// TIA Portal V18 program export: 1 tag tables, 7 data types, 4 data blocks, 9 code blocks (in call order from the OBs), 2 instance data blocks

VAR_GLOBAL   // PLC tag table "Default tag table"
   D_INPUT AT %I0.0 : "DI";
   A_IN AT %I100.0 : "AI";
   RTD_IN AT %I108.0 : "RTD";
   D_OUTPUT AT %Q0.0 : "DO";
   A_OUT AT %Q100.0 : "AO";
   System_Byte AT %MB1 : Byte;
   FirstScan AT %M1.0 : Bool;
   DiagStatusUpdate AT %M1.1 : Bool;
   AlwaysTRUE AT %M1.2 : Bool;
   AlwaysFALSE AT %M1.3 : Bool;
   Clock_Byte AT %MB0 : Byte;
   Clock_10Hz AT %M0.0 : Bool;
   Clock_5Hz AT %M0.1 : Bool;
   "Clock_2.5Hz" AT %M0.2 : Bool;
   Clock_2Hz AT %M0.3 : Bool;
   "Clock_1.25Hz" AT %M0.4 : Bool;
   Clock_1Hz AT %M0.5 : Bool;
   "Clock_0.625Hz" AT %M0.6 : Bool;
   "Clock_0.5Hz" AT %M0.7 : Bool;
   Tag_1 AT %M5.0 : Bool;
   Tag_2 AT %M55.0 : Bool;
   Tag_3 AT %M75.0 : Bool;
END_VAR
VAR_GLOBAL CONSTANT   // user constants
   "None(2)" : Pip := 65535;
   "Automatic update(2)" : Pip := 0;
   "PIP 1(2)" : Pip := 1;
   "PIP 2(2)" : Pip := 2;
   "PIP 3(2)" : Pip := 3;
   "PIP 4(2)" : Pip := 4;
   "PIP 5" : Pip := 5;
   "PIP 6" : Pip := 6;
   "PIP 7" : Pip := 7;
   "PIP 8" : Pip := 8;
   "PIP 9" : Pip := 9;
   "PIP 10" : Pip := 10;
   "PIP 11" : Pip := 11;
   "PIP 12" : Pip := 12;
   "PIP 13" : Pip := 13;
   "PIP 14" : Pip := 14;
   "PIP 15" : Pip := 15;
   "PIP 16" : Pip := 16;
   "PIP 17" : Pip := 17;
   "PIP 18" : Pip := 18;
   "PIP 19" : Pip := 19;
   "PIP 20" : Pip := 20;
   "PIP 21" : Pip := 21;
   "PIP 22" : Pip := 22;
   "PIP 23" : Pip := 23;
   "PIP 24" : Pip := 24;
   "PIP 25" : Pip := 25;
   "PIP 26" : Pip := 26;
   "PIP 27" : Pip := 27;
   "PIP 28" : Pip := 28;
   "PIP 29" : Pip := 29;
   "PIP 30" : Pip := 30;
   "PIP 31" : Pip := 31;
   "PIP OB Servo(2)" : Pip := 32768;
   "Local~MC(2)" : Hw_SubModule := 51;
   "Local~Common(2)" : Hw_SubModule := 50;
   "Local~Device(2)" : Hw_Device := 32;
   "Local~Configuration(2)" : Hw_SubModule := 33;
   "Local~Display" : Hw_SubModule := 54;
   "Local~Exec(2)" : Hw_SubModule := 52;
   "Local(2)" : Hw_SubModule := 49;
   "Local~PROFINET_interface_1(2)" : Hw_Interface := 64;
   "Local~PROFINET_interface_1~Port_1(2)" : Hw_Interface := 65;
   "Local~PROFINET_interface_1~Port_2" : Hw_Interface := 66;
   "Local~Virtual_communication_interface" : Hw_Interface := 135;
   "Local~License_Manager" : Hw_SubModule := 42;
   "OB_Main(2)" : OB_PCYCLE := 1;
END_VAR

TYPE "AI"
// stored: IsFailsafeCompliant false
   STRUCT
      "FLOW METER" : Int;
      "CONDUCTIVITY METER" : Int;
      "SPARE AI1" : Int;
      "SPARE AI2" : Int;
   END_STRUCT;
END_TYPE

TYPE "AM CTRL"
// stored: IsFailsafeCompliant false
   STRUCT
      "AUTO/MAN" : Bool := TRUE;
      "MAN START" : Bool;
      "MAN STOP" : Bool;
   END_STRUCT;
END_TYPE

TYPE "AO"
// stored: IsFailsafeCompliant false
   STRUCT
      VFD : Int;
      "SPARE AO" : Int;
   END_STRUCT;
END_TYPE

TYPE "DI"
// stored: IsFailsafeCompliant false
   STRUCT
      START : Bool;
      STOP : Bool;
      EMERGENCY : Bool;
      ACKNOWLEDGE : Bool;
      "AUTO/MANUAL" : Bool;
      "RECUPARATION TANK HL" : Bool;
      "RECUPARATION TANK LL" : Bool;
      "HOT WATER TANK HL" : Bool;
      "HOT WATER TANK LL" : Bool;
      "CAUSTIC TANK HL" : Bool;
      "CAUSTIC TANK LL" : Bool;
      "ACID TANK HL" : Bool;
      "ACID TANK LL" : Bool;
      "SUPPLY PUMP RUN (VFD)" : Bool;
      RESERVED : Bool;
      RESERVED_1 : Bool;
      "SUPPLY PUMP TRIP (VFD)" : Bool;
      "ACID DOSING PUMP RUN" : Bool;
      "ACID DOSING PUMP TRIP" : Bool;
      "CAUSTIC DOSING PUMP RUN" : Bool;
      "CAUSTIC DOSING PUMP TRIP" : Bool;
      "RETURN PUMP 1 RUN" : Bool;
      "RETURN PUMP 1 TRIP" : Bool;
      "RETURN PUMP 2 RUN" : Bool;
      "RETURN PUMP 2 TRIP" : Bool;
      "RETURN PUMP 3 RUN" : Bool;
      "RETURN PUMP 3 TRIP" : Bool;
      "FLOW SWITCH" : Bool;
      "PRESSURE SWITCH" : Bool;
      SPARE_1 : Bool;
      SPARE_2 : Bool;
      SPARE_3 : Bool;
   END_STRUCT;
END_TYPE

TYPE "DO"
// stored: IsFailsafeCompliant false
   STRUCT
      BUZZER : Bool;
      "BFV 1" : Bool;
      "BFV 2" : Bool;
      "BFV 3" : Bool;
      "BFV 4" : Bool;
      "BFV 5" : Bool;
      "BFV 6" : Bool;
      "BFV 7" : Bool;
      "BFV 8" : Bool;
      "BFV 9" : Bool;
      R1 : Bool;
      R2 : Bool;
      R3 : Bool;
      R4 : Bool;
      R5 : Bool;
      R6 : Bool;
      "BFV 10" : Bool;
      "BFV 11" : Bool;
      "BFV 12" : Bool;
      "BFV 13" : Bool;
      "BFV 14" : Bool;
      "BFV 15" : Bool;
      "BFV 16" : Bool;
      "BFV 17" : Bool;
      "BFV 18" : Bool;
      "BFV 19" : Bool;
      "CIP SUPPLY PUMP START (VFD)" : Bool;
      "ACID DOSING PUMP" : Bool;
      "CAUSTIC DOSING PUMP" : Bool;
      "RETURN PUMP 1" : Bool;
      "RETURN PUMP 2" : Bool;
      "RETUEN PUMP 3" : Bool;
   END_STRUCT;
END_TYPE

TYPE "RTD"
// stored: IsFailsafeCompliant false
   STRUCT
      "RECUPERATION TANK" : Int;
      "HOT WATER TANK" : Int;
      "CAUSTIC TANK" : Int;
      "ACID TANK" : Int;
      "FWD LINE" : Int;
      "RETURN LINE" : Int;
      "SPARE RTD" : Int;
      "SPARE RTD 1" : Int;
   END_STRUCT;
END_TYPE

TYPE "TANK DATA"
// stored: IsFailsafeCompliant false
   STRUCT
      "TANK TEMP SP" : Real;
      "LINE TEMP SP" : Real;
      "RETURN SP" : Real;
      "COND SP" : Real;
      "HYSTERIRIS TEMP" : Real;
      "HYSTERISIS COND" : Real;
      "CYCLE TIME MIN" : Int;
      "CYCLE TIME SEC" : Int;
      "ELAPSED MIN" : Int;
      "ELAPSED SEC" : Int;
   END_STRUCT;
END_TYPE

DATA_BLOCK "HMI ALARM DB"   // DB5
{ S7_Optimized_Access := 'FALSE' }
VERSION : 0.1
// stored: AutoNumber true, DBAccessibleFromOPCUA true, IsOnlyStoredInLoadMemory false, IsWriteProtectedInAS false
   VAR
      "FEED PUMP" : Byte;   // XO- INTERLOCK
      "ACID DOSING" : Byte;   // X1 - TRIP
      "CAUSTIC DOSING" : Byte;   // X2 - RUN FB ERROR
      "RP 1" : Byte;
      "RP 2" : Byte;
      "RP 3" : Byte;
      "RETURN NOT SELECTED" : Bool;
      "CYCLE NOT SELECTED" : Bool;
      "WATER FLUSH TIME NOT SET" : Bool;
      "HOT WATER TIME NOT SET" : Bool;
      "RECUP TIME NOT SET" : Bool;
      "ACIDIC TIME NOT SET" : Bool;
      "CAUSTIC TIMENOT SET" : Bool;
   END_VAR
BEGIN
END_DATA_BLOCK

DATA_BLOCK "HMI DB"   // DB2
{ S7_Optimized_Access := 'FALSE' }
VERSION : 0.1
// stored: AutoNumber true, DBAccessibleFromOPCUA true, IsOnlyStoredInLoadMemory false, IsWriteProtectedInAS false
   VAR RETAIN
      "START PREP" : Bool := FALSE;
      "START CIP" : Bool := FALSE;
      "CIP 3 STEP" : Bool := FALSE;
      "CIP 5 STEP" : Bool := FALSE;
      "CIP 7 STEP" : Bool := FALSE;
      RP1 : Bool;
      RP2 : Bool;
      RP3 : Bool;
      "RESUME CIP" : Bool;
      "RP1 SELECTED" : Bool;
      "RP2 SELECTED" : Bool;
      "RP3 SELECTED" : Bool;
      "3 STEP STATUS" : Word;
      "5 STEP STATUS" : Word;
      "9 STEP STATUS" : Word;
      RESERVE : Array[0..28] of Word;
      "BFV1 AM" { S7_SetPoint := 'True'} : "AM CTRL";
      "BFV2 AM" { S7_SetPoint := 'True'} : "AM CTRL";
      "BFV3 AM" { S7_SetPoint := 'True'} : "AM CTRL";
      "BFV4 AM" { S7_SetPoint := 'True'} : "AM CTRL";
      "BFV5 AM" { S7_SetPoint := 'True'} : "AM CTRL";
      "BFV6 AM" { S7_SetPoint := 'True'} : "AM CTRL";
      "BFV7 AM" { S7_SetPoint := 'True'} : "AM CTRL";
      "BFV8 AM" { S7_SetPoint := 'True'} : "AM CTRL";
      "BFV9 AM" { S7_SetPoint := 'True'} : "AM CTRL";
      "BFV10 AM" { S7_SetPoint := 'True'} : "AM CTRL";
      "BFV11 AM" { S7_SetPoint := 'True'} : "AM CTRL";
      "BFV12 AM" { S7_SetPoint := 'True'} : "AM CTRL";
      "BFV13 AM" { S7_SetPoint := 'True'} : "AM CTRL";
      "BFV14 AM" { S7_SetPoint := 'True'} : "AM CTRL";
      "BFV15 AM" { S7_SetPoint := 'True'} : "AM CTRL";
      "BFV16 AM" { S7_SetPoint := 'True'} : "AM CTRL";
      "BFV17 AM" { S7_SetPoint := 'True'} : "AM CTRL";
      "BFV18 AM" { S7_SetPoint := 'True'} : "AM CTRL";
      "BFV19 AM" { S7_SetPoint := 'True'} : "AM CTRL";
      "VFD AM" { S7_SetPoint := 'True'} : "AM CTRL";
      "RETURN PUMP 1 AM" { S7_SetPoint := 'True'} : "AM CTRL";
      "RETURN PUMP 2 AM" { S7_SetPoint := 'True'} : "AM CTRL";
      "RETURN PUMP 3 AM" { S7_SetPoint := 'True'} : "AM CTRL";
      "CAUSTIC AM" { S7_SetPoint := 'True'} : "AM CTRL";
      "ACIDIC AM" { S7_SetPoint := 'True'} : "AM CTRL";
      "PUMP SLOW SP" : Int := 0;
      RECUP : "TANK DATA";
      "HOT WATER" : "TANK DATA";
      CAUSTIC : "TANK DATA";
      ACIDIC : "TANK DATA";
      "ANALOG VALUES" : Struct
         FLOW : Real := 0.0;
         CONDCTIVITY : Real := 0.0;
         "RECUP TEMP" : Real := 0.0;
         "HOT WTR TEMP" : Real := 0.0;
         "CAUSTIC TEMP" : Real := 0.0;
         "ACID TEMP" : Real := 0.0;
         "RETURN LINE TEMP" : Real := 0.0;
      END_STRUCT;
      "START DELAYS" : Struct
         "RP1 MIN" : Int;
         "RP1 SEC" : Int;
         "RP2 MIN" : Int;
         "RP2 SEC" : Int;
         "RP3 MIN" : Int;
         "RP3 SEC" : Int;
      END_STRUCT;
      "COMMON SETPOINTS" : Struct   // 286
         "COND MIN FOR RECUP" : Real;
         "TMP MIN FOR RECUP" : Real;
         "WATER FLUSH MIN" : Int;
         "WATER FLUSH SEC" : Int;
         "WATER FLUSH REM MIN" : Int;
         "WATER FLUSH REM SEC" : Int;
      END_STRUCT;
      "Fwd line temp" : Real;
   END_VAR
BEGIN
   "BFV1 AM"."AUTO/MAN" := TRUE;
   "BFV1 AM"."MAN START" := FALSE;
   "BFV1 AM"."MAN STOP" := FALSE;
   "BFV2 AM"."AUTO/MAN" := TRUE;
   "BFV2 AM"."MAN START" := FALSE;
   "BFV2 AM"."MAN STOP" := FALSE;
   "BFV3 AM"."AUTO/MAN" := TRUE;
   "BFV3 AM"."MAN START" := FALSE;
   "BFV3 AM"."MAN STOP" := FALSE;
   "BFV4 AM"."AUTO/MAN" := TRUE;
   "BFV4 AM"."MAN START" := FALSE;
   "BFV4 AM"."MAN STOP" := FALSE;
   "BFV5 AM"."AUTO/MAN" := TRUE;
   "BFV5 AM"."MAN START" := FALSE;
   "BFV5 AM"."MAN STOP" := FALSE;
   "BFV6 AM"."AUTO/MAN" := TRUE;
   "BFV6 AM"."MAN START" := FALSE;
   "BFV6 AM"."MAN STOP" := FALSE;
   "BFV7 AM"."AUTO/MAN" := TRUE;
   "BFV7 AM"."MAN START" := FALSE;
   "BFV7 AM"."MAN STOP" := FALSE;
   "BFV8 AM"."AUTO/MAN" := TRUE;
   "BFV8 AM"."MAN START" := FALSE;
   "BFV8 AM"."MAN STOP" := FALSE;
   "BFV9 AM"."AUTO/MAN" := TRUE;
   "BFV9 AM"."MAN START" := FALSE;
   "BFV9 AM"."MAN STOP" := FALSE;
   "BFV10 AM"."AUTO/MAN" := TRUE;
   "BFV10 AM"."MAN START" := FALSE;
   "BFV10 AM"."MAN STOP" := FALSE;
   "BFV11 AM"."AUTO/MAN" := TRUE;
   "BFV11 AM"."MAN START" := FALSE;
   "BFV11 AM"."MAN STOP" := FALSE;
   "BFV12 AM"."AUTO/MAN" := TRUE;
   "BFV12 AM"."MAN START" := FALSE;
   "BFV12 AM"."MAN STOP" := FALSE;
   "BFV13 AM"."AUTO/MAN" := TRUE;
   "BFV13 AM"."MAN START" := FALSE;
   "BFV13 AM"."MAN STOP" := FALSE;
   "BFV14 AM"."AUTO/MAN" := TRUE;
   "BFV14 AM"."MAN START" := FALSE;
   "BFV14 AM"."MAN STOP" := FALSE;
   "BFV15 AM"."AUTO/MAN" := TRUE;
   "BFV15 AM"."MAN START" := FALSE;
   "BFV15 AM"."MAN STOP" := FALSE;
   "BFV16 AM"."AUTO/MAN" := TRUE;
   "BFV16 AM"."MAN START" := FALSE;
   "BFV16 AM"."MAN STOP" := FALSE;
   "BFV17 AM"."AUTO/MAN" := TRUE;
   "BFV17 AM"."MAN START" := FALSE;
   "BFV17 AM"."MAN STOP" := FALSE;
   "BFV18 AM"."AUTO/MAN" := TRUE;
   "BFV18 AM"."MAN START" := FALSE;
   "BFV18 AM"."MAN STOP" := FALSE;
   "BFV19 AM"."AUTO/MAN" := TRUE;
   "BFV19 AM"."MAN START" := FALSE;
   "BFV19 AM"."MAN STOP" := FALSE;
   "VFD AM"."AUTO/MAN" := TRUE;
   "VFD AM"."MAN START" := FALSE;
   "VFD AM"."MAN STOP" := FALSE;
   "RETURN PUMP 1 AM"."AUTO/MAN" := TRUE;
   "RETURN PUMP 1 AM"."MAN START" := FALSE;
   "RETURN PUMP 1 AM"."MAN STOP" := FALSE;
   "RETURN PUMP 2 AM"."AUTO/MAN" := TRUE;
   "RETURN PUMP 2 AM"."MAN START" := FALSE;
   "RETURN PUMP 2 AM"."MAN STOP" := FALSE;
   "RETURN PUMP 3 AM"."AUTO/MAN" := TRUE;
   "RETURN PUMP 3 AM"."MAN START" := FALSE;
   "RETURN PUMP 3 AM"."MAN STOP" := FALSE;
   "CAUSTIC AM"."AUTO/MAN" := TRUE;
   "CAUSTIC AM"."MAN START" := FALSE;
   "CAUSTIC AM"."MAN STOP" := FALSE;
   "ACIDIC AM"."AUTO/MAN" := TRUE;
   "ACIDIC AM"."MAN START" := FALSE;
   "ACIDIC AM"."MAN STOP" := FALSE;
   RECUP."COND SP" := 0.0;
   RECUP."HYSTERIRIS TEMP" := 0.0;
   RECUP."HYSTERISIS COND" := 0.0;
   RECUP."CYCLE TIME SEC" := 0;
   RECUP."ELAPSED MIN" := 0;
   RECUP."ELAPSED SEC" := 0;
   "HOT WATER"."COND SP" := 0.0;
   "HOT WATER"."HYSTERIRIS TEMP" := 0.0;
   "HOT WATER"."HYSTERISIS COND" := 0.0;
   "HOT WATER"."CYCLE TIME MIN" := 0;
   "HOT WATER"."CYCLE TIME SEC" := 0;
   "HOT WATER"."ELAPSED MIN" := 0;
   "HOT WATER"."ELAPSED SEC" := 0;
   CAUSTIC."COND SP" := 0.0;
   CAUSTIC."HYSTERIRIS TEMP" := 0.0;
   CAUSTIC."HYSTERISIS COND" := 0.0;
   CAUSTIC."CYCLE TIME MIN" := 0;
   CAUSTIC."CYCLE TIME SEC" := 0;
   CAUSTIC."ELAPSED MIN" := 0;
   CAUSTIC."ELAPSED SEC" := 0;
   ACIDIC."COND SP" := 0.0;
   ACIDIC."HYSTERIRIS TEMP" := 0.0;
   ACIDIC."HYSTERISIS COND" := 0.0;
   ACIDIC."CYCLE TIME MIN" := 0;
   ACIDIC."CYCLE TIME SEC" := 0;
   ACIDIC."ELAPSED MIN" := 0;
   ACIDIC."ELAPSED SEC" := 0;
END_DATA_BLOCK

DATA_BLOCK "IO_MAP"   // DB1
{ S7_Optimized_Access := 'FALSE' }
VERSION : 0.1
// stored: AutoNumber true, DBAccessibleFromOPCUA true, IsOnlyStoredInLoadMemory false, IsWriteProtectedInAS false
   VAR
      D_IN { S7_SetPoint := 'True'} : "DI";
      D_OUT { S7_SetPoint := 'True'} : "DO";
      A_OUT { S7_SetPoint := 'True'} : "AO";
      A_IN { S7_SetPoint := 'True'} : "AI";
      RTD { S7_SetPoint := 'True'} : "RTD";
   END_VAR
BEGIN
END_DATA_BLOCK

DATA_BLOCK "OPERATIONS DB"   // DB3
{ S7_Optimized_Access := 'TRUE' }
VERSION : 0.1
// stored: AutoNumber true, DBAccessibleFromOPCUA true, IsOnlyStoredInLoadMemory false, IsRetainMemResEnabled false, IsWriteProtectedInAS false, MemoryReserve 100
   VAR
      "SYSTEM STARTED" : Bool;
   END_VAR
BEGIN
END_DATA_BLOCK

ORGANIZATION_BLOCK "Main"   // OB1, LAD, ProgramCycle
TITLE = "Main Program Sweep (Cycle)"
{ S7_Optimized_Access := 'TRUE' }
VERSION : 0.1
// stored: AutoNumber true, IsIECCheckEnabled false, SetENOAutomatically false
   VAR_INPUT
      Initial_Call : Bool;   // Initial call of this OB
      Remanence : Bool;   // =True, if remanent data are available
   END_VAR
   VAR_TEMP   // added for the SCL form of the ladder/FBD networks
      _w1 : Bool;
   END_VAR
BEGIN

REGION Network 1
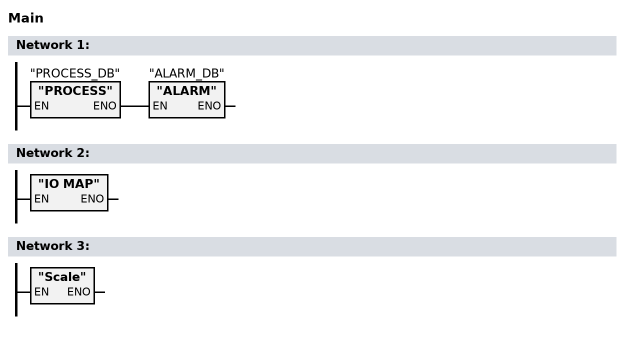
   RUNG wire#powerrail
      "PROCESS_DB"()
      "ALARM_DB"()
   END_RUNG
   // the same network as SCL:
   "PROCESS_DB"(ENO => #_w1);   // "PROCESS"
   IF #_w1 THEN
       "ALARM_DB"();   // "ALARM"
   END_IF;
END_REGION

REGION Network 2
   RUNG wire#powerrail
      "IO MAP"()
   END_RUNG
   // the same network as SCL:
   "IO MAP"();
END_REGION

REGION Network 3
   RUNG wire#powerrail
      "Scale"()
   END_RUNG
   // the same network as SCL:
   "Scale"();
END_REGION
END_ORGANIZATION_BLOCK

FUNCTION_BLOCK "PROCESS"   // FB3, LAD
{ S7_Optimized_Access := 'TRUE' }
VERSION : 0.1
// stored: AutoNumber true, IsIECCheckEnabled false, IsRetainMemResEnabled false, MemoryReserve 100, SetENOAutomatically false, UDAEnableTagReadback false
   VAR
      "RECUP TANK" { S7_SetPoint := 'True'} : "TANK";
      "HOT WATER TANK" { S7_SetPoint := 'True'} : "TANK";
      "CAUSTIC TANK" { S7_SetPoint := 'True'} : "TANK";
      "ACID TANK" { S7_SetPoint := 'True'} : "TANK";
      "RECUP PREP DONE" { S7_SetPoint := 'True'} : Bool;
      "HOT WTR PREP DONE" : Bool;
      "CAUSTIC PREP DONE" : Bool;
      "ACID PREP DONE" : Bool;
      "PREP FINISHED PULSE" : Bool;
      P1 : Bool;
      P2 : Bool;
      P3 : Bool;
      P4 : Bool;
      P5 : Bool;
      P6 : Bool;
      P7 : Bool;
      P8 : Bool;
      P9 : Bool;
      P10 : Bool;
      CIP_STARTED : Bool;
      "3 CIP FINISH PULSE" : Bool;
      "5 CIP FINISH PULSE" : Bool;
      "7 CIP FINISH PULSE" : Bool;
      "PUMP OK" : Bool;
   END_VAR
   VAR RETAIN
      "RECUP CIP DONE" : Array[0..4] of Bool;
      "HOT WTR CIP DONE" : Array[0..4] of Bool;
      "CAUSTIC CIP DONE" : Array[0..4] of Bool;
      "ACID CIP DONE" : Array[0..4] of Bool;
      "WATER FLUSH CIP DONE" : Array[0..4] of Bool;
      "CIP_STEP SELECTED" : Int;
   END_VAR
   VAR
      "CURCULATION PUMP" { S7_SetPoint := 'True'} : "PUMP";
      "BFV1 CTRL" { S7_SetPoint := 'True'} : "VALVE CTRL";
      "BFV2 CTRL" { S7_SetPoint := 'True'} : "VALVE CTRL";
      "BFV3 CTRL" { S7_SetPoint := 'True'} : "VALVE CTRL";
      "BFV4 CTRL" { S7_SetPoint := 'True'} : "VALVE CTRL";
      "BFV5 CTRL" { S7_SetPoint := 'True'} : "VALVE CTRL";
      "BFV6 CTRL" { S7_SetPoint := 'True'} : "VALVE CTRL";
      "BFV7 CTRL" { S7_SetPoint := 'True'} : "VALVE CTRL";
      "BFV8 CTRL" { S7_SetPoint := 'True'} : "VALVE CTRL";
      "BFV9 CTRL" { S7_SetPoint := 'True'} : "VALVE CTRL";
      "BFV10 CTRL" { S7_SetPoint := 'True'} : "VALVE CTRL";
      "BFV11 CTRL" { S7_SetPoint := 'True'} : "VALVE CTRL";
      "BFV12 CTRL" { S7_SetPoint := 'True'} : "VALVE CTRL";
      "BFV13 CTRL" { S7_SetPoint := 'True'} : "VALVE CTRL";
      "BFV14 CTRL" { S7_SetPoint := 'True'} : "VALVE CTRL";
      "BFV15 CTRL" { S7_SetPoint := 'True'} : "VALVE CTRL";
      "BFV16 CTRL" { S7_SetPoint := 'True'} : "VALVE CTRL";
      "BFV17 CTRL" { S7_SetPoint := 'True'} : "VALVE CTRL";
      "BFV18 CTRL" { S7_SetPoint := 'True'} : "VALVE CTRL";
      "BFV19 CTRL" { S7_SetPoint := 'True'} : "VALVE CTRL";
      "BFV20 CTRL" { S7_SetPoint := 'True'} : "VALVE CTRL";
      "CAUSTIC DOSING" { S7_SetPoint := 'True'} : "PUMP";
      "ACID DOSING" { S7_SetPoint := 'True'} : "PUMP";
      "RETURN PUMP 1" { S7_SetPoint := 'True'} : "PUMP";
      "RETURN PUMP 2" { S7_SetPoint := 'True'} : "PUMP";
      "RETURN PUMP 3" { S7_SetPoint := 'True'} : "PUMP";
      "WATER FLUSH" { S7_SetPoint := 'True'} : TON_TIME;
   END_VAR
   VAR_TEMP
      "RECUP PREP START" : Bool;
      "RECUP CIP START" : Bool;
      "HOT WTR PREP START" : Bool;
      "HOT WTR CIP START" : Bool;
      "CAUSTIC PREP START" : Bool;
      "CAUSTIC CIP START" : Bool;
      "ACID PREP START" : Bool;
      "ACID CIP START" : Bool;
      "WATER FLUSH CIP START" : Bool;
      "RP1 START" : Bool;
      "RP2 START" : Bool;
      "RP3 START" : Bool;
      CIRCULATION : Bool;
      "WF PT" : Time;
      "WF ET" : Time;
      RECUP : Struct
         "INLET 1 OPEN" : Bool;
         "INLET 2 OPEN" : Bool;
         "OUTLE OPEN" : Bool;
         "START DOZING" : Bool;
         FLUSH : Bool;
         HEATING : Bool;
         "PREP DONE" : Bool;
      END_STRUCT;
      HTWTR : Struct
         "INLET 1 OPEN" : Bool;
         "INLET 2 OPEN" : Bool;
         "OUTLE OPEN" : Bool;
         "START DOZING" : Bool;
         FLUSH : Bool;
         HEATING : Bool;
         "PREP DONE" : Bool;
      END_STRUCT;
      CAUSTIC : Struct
         "INLET 1 OPEN" : Bool;
         "INLET 2 OPEN" : Bool;
         "OUTLE OPEN" : Bool;
         "START DOZING" : Bool;
         FLUSH : Bool;
         HEATING : Bool;
         "PREP DONE" : Bool;
      END_STRUCT;
      ACIDIC : Struct
         "INLET 1 OPEN" : Bool;
         "INLET 2 OPEN" : Bool;
         "OUTLE OPEN" : Bool;
         "START DOZING" : Bool;
         FLUSH : Bool;
         HEATING : Bool;
         "PREP DONE" : Bool;
      END_STRUCT;
      "TEMP ARRAY" : Array[0..4] of Bool;
      "CYCLE SELECTED" : Bool;
      "RETURN SELECTED" : Bool;
      "settings OK" : Bool;
      "WATER TIME OK" : Bool;
      "CAUSTIC TIME OK" : Bool;
      "HOTWATER TIME OK" : Bool;
      "REUP TIME OK" : Bool;
      "ACID TIME OK" : Bool;
   END_VAR
   VAR_TEMP   // added for the SCL form of the ladder/FBD networks
      _w1 : Bool;
      _w2 : Bool;
      _w3 : Bool;
      _w4 : Bool;
      _w5 : Bool;
      _w6 : Bool;
      _w7 : Bool;
      _w8 : Bool;
      _w9 : Bool;
      _w10 : Bool;
   END_VAR
BEGIN

REGION Network 1: START PREP
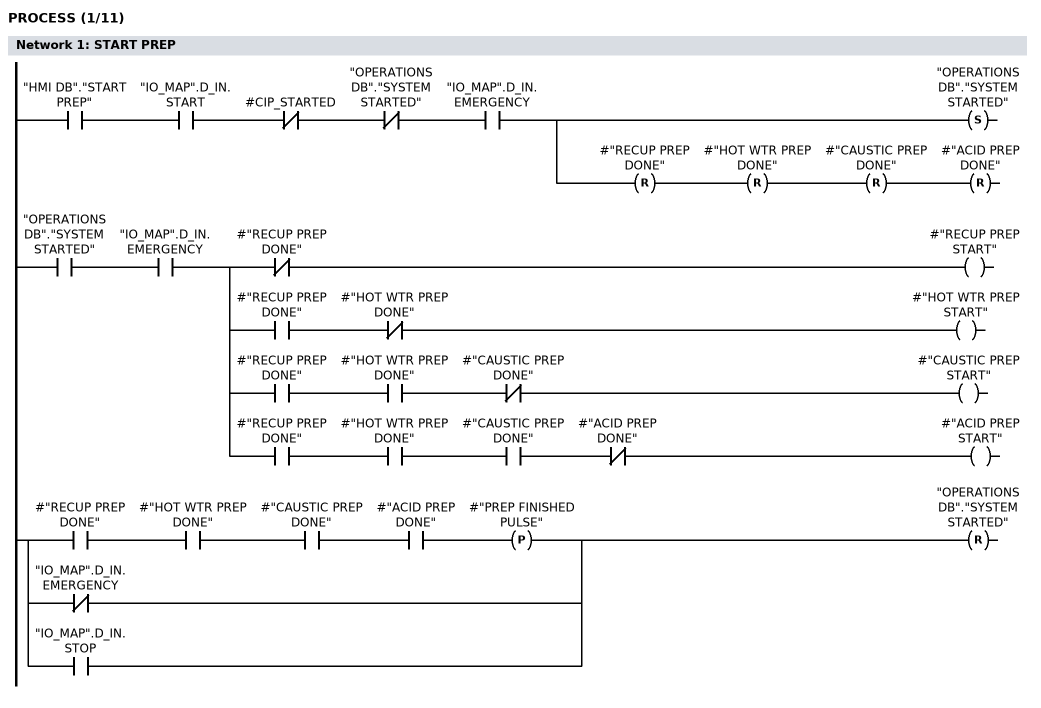
   RUNG wire#powerrail
      Contact( "HMI DB"."START PREP" )
      Contact( "IO_MAP".D_IN.START )
      I_Contact( #CIP_STARTED )
      I_Contact( "OPERATIONS DB"."SYSTEM STARTED" )
      Contact( "IO_MAP".D_IN.EMERGENCY )
      wire#w1
      S_Coil( "OPERATIONS DB"."SYSTEM STARTED" )
   END_RUNG
   RUNG wire#w1
      R_Coil( #"RECUP PREP DONE" )
      R_Coil( #"HOT WTR PREP DONE" )
      R_Coil( #"CAUSTIC PREP DONE" )
      R_Coil( #"ACID PREP DONE" )
   END_RUNG
   RUNG wire#powerrail
      Contact( "OPERATIONS DB"."SYSTEM STARTED" )
      Contact( "IO_MAP".D_IN.EMERGENCY )
      wire#w2
      I_Contact( #"RECUP PREP DONE" )
      Coil( #"RECUP PREP START" )
   END_RUNG
   RUNG wire#w2
      Contact( #"RECUP PREP DONE" )
      I_Contact( #"HOT WTR PREP DONE" )
      Coil( #"HOT WTR PREP START" )
   END_RUNG
   RUNG wire#w2
      Contact( #"RECUP PREP DONE" )
      Contact( #"HOT WTR PREP DONE" )
      I_Contact( #"CAUSTIC PREP DONE" )
      Coil( #"CAUSTIC PREP START" )
   END_RUNG
   RUNG wire#w2
      Contact( #"RECUP PREP DONE" )
      Contact( #"HOT WTR PREP DONE" )
      Contact( #"CAUSTIC PREP DONE" )
      I_Contact( #"ACID PREP DONE" )
      Coil( #"ACID PREP START" )
   END_RUNG
   RUNG wire#powerrail
      Contact( #"RECUP PREP DONE" )
      Contact( #"HOT WTR PREP DONE" )
      Contact( #"CAUSTIC PREP DONE" )
      Contact( #"ACID PREP DONE" )
      P_Trig( #"PREP FINISHED PULSE" )
      wire#w3
      R_Coil( "OPERATIONS DB"."SYSTEM STARTED" )
   END_RUNG
   RUNG wire#powerrail
      I_Contact( "IO_MAP".D_IN.EMERGENCY )
   END_RUNG wire#w3
   RUNG wire#powerrail
      Contact( "IO_MAP".D_IN.STOP )
   END_RUNG wire#w3
   // the same network as SCL:
   #_w1 := "HMI DB"."START PREP" AND "IO_MAP".D_IN.START AND NOT #CIP_STARTED AND NOT "OPERATIONS DB"."SYSTEM STARTED" AND "IO_MAP".D_IN.EMERGENCY;
   IF #_w1 THEN
       "OPERATIONS DB"."SYSTEM STARTED" := TRUE;
       #"RECUP PREP DONE" := FALSE;
       #"HOT WTR PREP DONE" := FALSE;
       #"CAUSTIC PREP DONE" := FALSE;
       #"ACID PREP DONE" := FALSE;
   END_IF;
   #_w2 := "OPERATIONS DB"."SYSTEM STARTED" AND "IO_MAP".D_IN.EMERGENCY;
   #"RECUP PREP START" := #_w2 AND NOT #"RECUP PREP DONE";
   #"HOT WTR PREP START" := #_w2 AND #"RECUP PREP DONE" AND NOT #"HOT WTR PREP DONE";
   #"CAUSTIC PREP START" := #_w2 AND #"RECUP PREP DONE" AND #"HOT WTR PREP DONE" AND NOT #"CAUSTIC PREP DONE";
   #"ACID PREP START" := #_w2 AND #"RECUP PREP DONE" AND #"HOT WTR PREP DONE" AND #"CAUSTIC PREP DONE" AND NOT #"ACID PREP DONE";
   #_w3 := #"RECUP PREP DONE" AND #"HOT WTR PREP DONE" AND #"CAUSTIC PREP DONE" AND #"ACID PREP DONE";
   #_w4 := #_w3 AND NOT #"PREP FINISHED PULSE";   // rising edge
   #"PREP FINISHED PULSE" := #_w3;
   IF #_w4 OR NOT "IO_MAP".D_IN.EMERGENCY OR "IO_MAP".D_IN.STOP THEN
       "OPERATIONS DB"."SYSTEM STARTED" := FALSE;
   END_IF;
END_REGION

REGION Network 2 (SCL): START CIP
   //check for settings if it is ok to procced with CIP steps
   #"CYCLE SELECTED" := "HMI DB"."CIP 3 STEP" OR "HMI DB"."CIP 5 STEP" OR "HMI DB"."CIP 7 STEP";
   #"RETURN SELECTED" := "HMI DB"."RP1 SELECTED" OR "HMI DB"."RP2 SELECTED" OR "HMI DB"."RP3 SELECTED";
   #"WATER TIME OK" := ("HMI DB"."COMMON SETPOINTS"."WATER FLUSH MIN" > 0 OR "HMI DB"."COMMON SETPOINTS"."WATER FLUSH SEC" > 0);
   #"REUP TIME OK" := ("HMI DB".RECUP."CYCLE TIME MIN" > 0 OR "HMI DB".RECUP."CYCLE TIME SEC" > 0);
   #"HOTWATER TIME OK" := ("HMI DB"."HOT WATER"."CYCLE TIME MIN" > 0 OR "HMI DB"."HOT WATER"."CYCLE TIME SEC" > 0);
   #"CAUSTIC TIME OK" := ("HMI DB".CAUSTIC."CYCLE TIME MIN" > 0 OR "HMI DB".CAUSTIC."CYCLE TIME SEC" > 0) OR "HMI DB"."CIP 3 STEP";
   #"ACID TIME OK" := ("HMI DB".ACIDIC ."CYCLE TIME MIN" > 0 OR "HMI DB".ACIDIC."CYCLE TIME SEC" > 0) OR "HMI DB"."CIP 3 STEP" OR "HMI DB"."CIP 5 STEP" ;

   #"settings OK" := #"CYCLE SELECTED" AND #"RETURN SELECTED" AND #"WATER TIME OK" AND #"REUP TIME OK" AND #"HOTWATER TIME OK" AND #"CAUSTIC TIME OK" AND #"ACID TIME OK";
   //IF SETTINGS ARE OK STARTING CONDITIONS FOR CIP CYCLE
   IF ("HMI DB"."START CIP" OR "HMI DB"."RESUME CIP") AND"IO_MAP".D_IN.START AND"IO_MAP".D_IN.EMERGENCY AND NOT"OPERATIONS DB"."SYSTEM STARTED"AND NOT #CIP_STARTED AND NOT"IO_MAP".D_IN.STOP  AND #"settings OK" THEN
       #CIP_STARTED := TRUE;
       IF "HMI DB"."CIP 3 STEP" THEN
           #"CIP_STEP SELECTED" := 3;
       ELSIF "HMI DB"."CIP 5 STEP" THEN
           #"CIP_STEP SELECTED" := 5;
       ELSIF "HMI DB"."CIP 7 STEP" THEN
           #"CIP_STEP SELECTED" := 9;
       END_IF;
       IF "HMI DB"."START CIP" THEN
           #"RECUP CIP DONE" := #"TEMP ARRAY";
           #"HOT WTR CIP DONE" := #"TEMP ARRAY";
           #"CAUSTIC CIP DONE" := #"TEMP ARRAY";
           #"ACID CIP DONE" := #"TEMP ARRAY";
           #"WATER FLUSH CIP DONE" := #"TEMP ARRAY";
       END_IF;

       //STOP CONDITION IF EMERGENCY OR STOP IS PRESSED
   ELSIF NOT "IO_MAP".D_IN.EMERGENCY OR "IO_MAP".D_IN.STOP  THEN
       #CIP_STARTED := FALSE;
        #"CIP_STEP SELECTED" := 0;
   END_IF;
END_REGION

REGION Network 3 (SCL): CIP SEQUENCE
   IF #CIP_STARTED THEN
       CASE #"CIP_STEP SELECTED" OF
               //SEQUENCE FOR 3 STEP OPERATION
           3:
               #"RECUP CIP START" := NOT #"RECUP CIP DONE"[0];
               #"HOT WTR CIP START" := #"RECUP CIP DONE"[0] AND NOT #"HOT WTR CIP DONE"[0];
               #"WATER FLUSH CIP START" := #"RECUP CIP DONE"[0] AND #"HOT WTR CIP DONE"[0] AND NOT #"WATER FLUSH CIP DONE"[0];

               //3 STEP DONE CONDITION
               IF #"RECUP CIP DONE"[0] AND #"HOT WTR CIP DONE"[0] AND #"WATER FLUSH CIP DONE"[0] AND NOT #"3 CIP FINISH PULSE" THEN
                   #CIP_STARTED := FALSE;
                   #"3 CIP FINISH PULSE" := TRUE;
               ELSIF NOT (#"RECUP CIP DONE"[0] AND #"HOT WTR CIP DONE"[0] AND #"WATER FLUSH CIP DONE"[0]) THEN
                   #"3 CIP FINISH PULSE" := FALSE;
               END_IF;
           5:
               //SEQUENCE FOR 5 STEP OPERATION
               #"RECUP CIP START" := NOT #"RECUP CIP DONE"[0];
               #"CAUSTIC CIP START" := #"RECUP CIP DONE"[0] AND NOT #"CAUSTIC CIP DONE"[0];
               #"WATER FLUSH CIP START" := (#"RECUP CIP DONE"[0] AND #"CAUSTIC CIP DONE"[0] AND NOT #"WATER FLUSH CIP DONE"[0])
               OR (#"RECUP CIP DONE"[0] AND #"CAUSTIC CIP DONE"[0] AND #"WATER FLUSH CIP DONE"[0] AND #"HOT WTR CIP DONE"[0] AND NOT #"WATER FLUSH CIP DONE"[1]);
               #"HOT WTR CIP START" := #"RECUP CIP DONE"[0] AND #"CAUSTIC CIP DONE"[0] AND #"WATER FLUSH CIP DONE"[0] AND NOT #"HOT WTR CIP DONE"[0];

               // 5 STEP DONE CONDITION
               IF #"RECUP CIP DONE"[0] AND #"CAUSTIC CIP DONE"[0] AND #"WATER FLUSH CIP DONE"[0] AND #"HOT WTR CIP DONE"[0] AND #"WATER FLUSH CIP DONE"[1] AND NOT #"5 CIP FINISH PULSE" THEN
                   #CIP_STARTED := FALSE;
                   #"5 CIP FINISH PULSE" := TRUE;
               ELSIF NOT (#"RECUP CIP DONE"[0] AND #"CAUSTIC CIP DONE"[0] AND #"WATER FLUSH CIP DONE"[0] AND #"HOT WTR CIP DONE"[0] AND #"WATER FLUSH CIP DONE"[1]) THEN
                   #"5 CIP FINISH PULSE" := FALSE;
               END_IF;

           9:
               //SEQUENCE FOR 9 STEP OPERATION
               #"RECUP CIP START" := NOT #"RECUP CIP DONE"[0];

               #"CAUSTIC CIP START" := (#"RECUP CIP DONE"[0] AND NOT #"CAUSTIC CIP DONE"[0])
               OR #"RECUP CIP DONE"[0] AND #"CAUSTIC CIP DONE"[0] AND #"WATER FLUSH CIP DONE"[0] AND #"ACID CIP DONE"[0] AND #"WATER FLUSH CIP DONE"[1] AND NOT #"CAUSTIC CIP DONE"[1];

               #"WATER FLUSH CIP START" := (#"RECUP CIP DONE"[0] AND #"CAUSTIC CIP DONE"[0] AND NOT #"WATER FLUSH CIP DONE"[0])
               OR (#"RECUP CIP DONE"[0] AND #"CAUSTIC CIP DONE"[0] AND #"WATER FLUSH CIP DONE"[0] AND #"ACID CIP DONE"[0] AND NOT #"WATER FLUSH CIP DONE"[1])
               OR (#"RECUP CIP DONE"[0] AND #"CAUSTIC CIP DONE"[0] AND #"WATER FLUSH CIP DONE"[0] AND #"ACID CIP DONE"[0] AND #"WATER FLUSH CIP DONE"[1] AND #"CAUSTIC CIP DONE"[1] AND NOT #"WATER FLUSH CIP DONE"[2])
               OR (#"RECUP CIP DONE"[0] AND #"CAUSTIC CIP DONE"[0] AND #"WATER FLUSH CIP DONE"[0] AND #"ACID CIP DONE"[0] AND  #"WATER FLUSH CIP DONE"[1] AND #"CAUSTIC CIP DONE"[1] AND #"WATER FLUSH CIP DONE"[2] AND #"HOT WTR CIP DONE"[0] AND NOT #"WATER FLUSH CIP DONE"[3]);

               #"ACID CIP START" := #"RECUP CIP DONE"[0] AND #"CAUSTIC CIP DONE"[0] AND #"WATER FLUSH CIP DONE"[0] AND NOT #"ACID CIP DONE"[0];

               #"HOT WTR CIP START" := (#"RECUP CIP DONE"[0] AND #"CAUSTIC CIP DONE"[0] AND #"WATER FLUSH CIP DONE"[0] AND #"ACID CIP DONE"[0] AND  #"WATER FLUSH CIP DONE"[1] AND #"CAUSTIC CIP DONE"[1] AND #"WATER FLUSH CIP DONE"[2] AND NOT #"HOT WTR CIP DONE"[0]);

               //9 STEP DONE
               IF #"RECUP CIP DONE"[0] AND #"CAUSTIC CIP DONE"[0] AND #"WATER FLUSH CIP DONE"[0] AND #"ACID CIP DONE"[0] AND  #"WATER FLUSH CIP DONE"[1] AND #"CAUSTIC CIP DONE"[1] AND #"WATER FLUSH CIP DONE"[2] AND #"HOT WTR CIP DONE"[0] AND #"WATER FLUSH CIP DONE"[3] AND NOT #"7 CIP FINISH PULSE" THEN
                   #CIP_STARTED := FALSE;
                   #"7 CIP FINISH PULSE" := TRUE;
               ELSIF NOT (#"RECUP CIP DONE"[0] AND #"CAUSTIC CIP DONE"[0] AND #"WATER FLUSH CIP DONE"[0] AND #"ACID CIP DONE"[0] AND NOT #"WATER FLUSH CIP DONE"[1] AND #"CAUSTIC CIP DONE"[1] AND #"WATER FLUSH CIP DONE"[2] AND #"HOT WTR CIP DONE"[0] AND #"WATER FLUSH CIP DONE"[3]) THEN
                   #"7 CIP FINISH PULSE" := FALSE;
               END_IF;
       END_CASE;
   END_IF;
END_REGION

REGION Network 4: RECUPARATION TANK
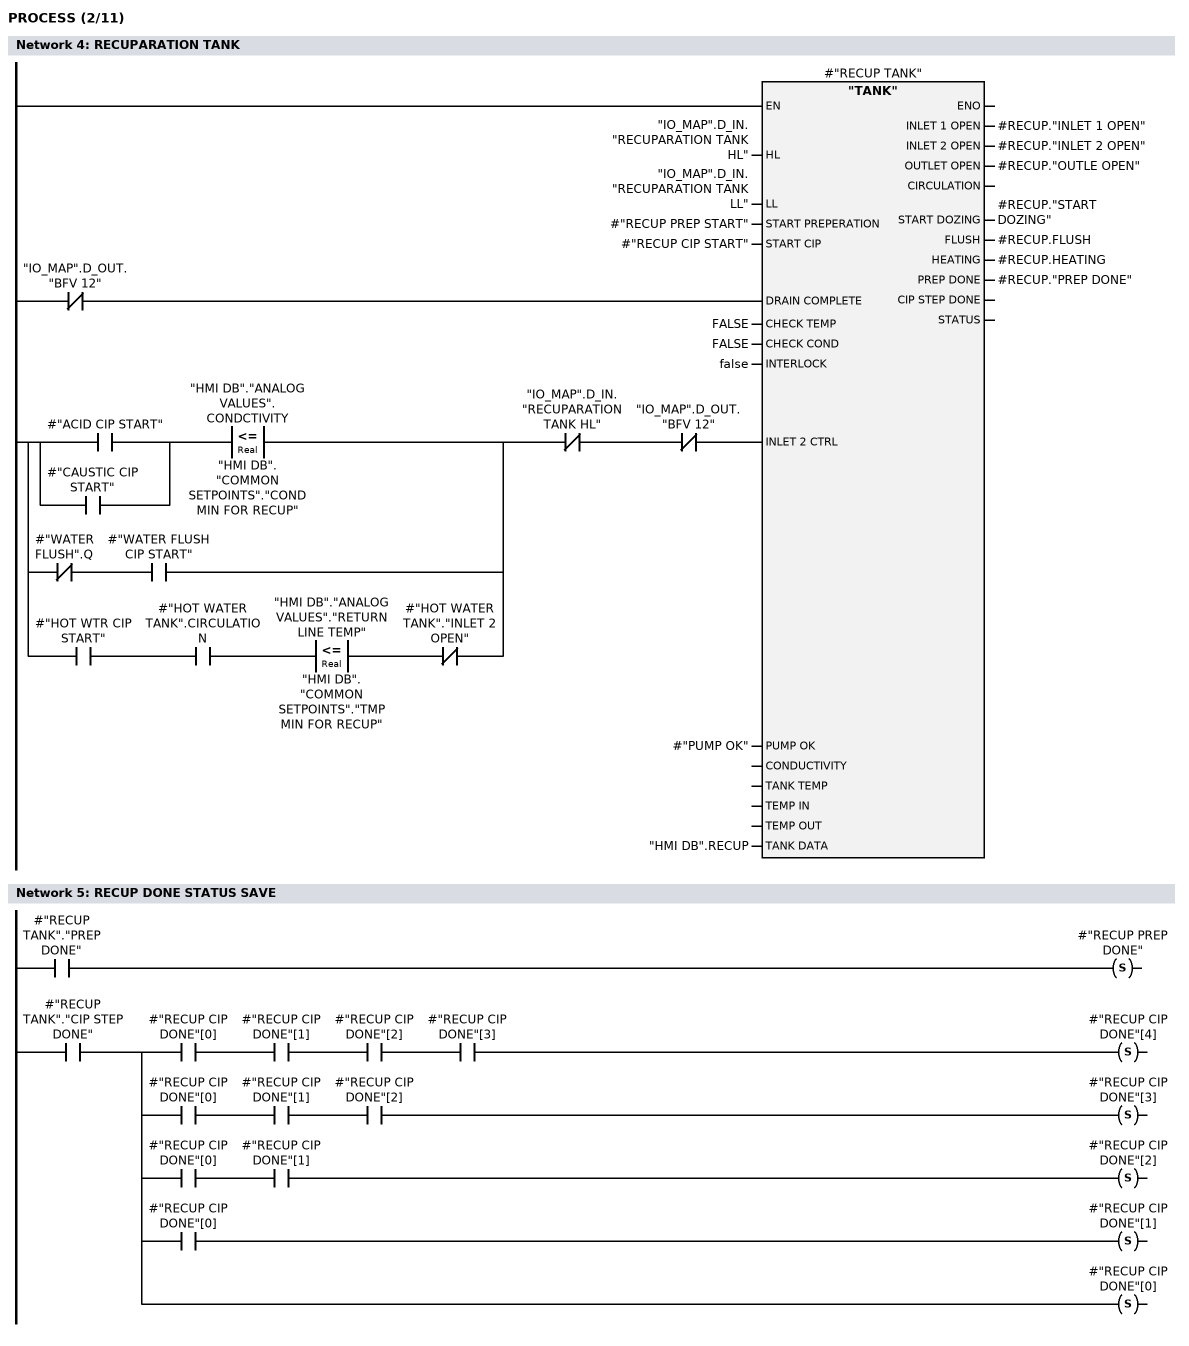
   RUNG wire#powerrail
      #"RECUP TANK"("DRAIN COMPLETE" := wire#w1, "INLET 2 CTRL" := wire#w4, HL := "IO_MAP".D_IN."RECUPARATION TANK HL", LL := "IO_MAP".D_IN."RECUPARATION TANK LL", "START PREPERATION" := #"RECUP PREP START", "START CIP" := #"RECUP CIP START", "CHECK TEMP" := FALSE, "CHECK COND" := FALSE, INTERLOCK := false, "PUMP OK" := #"PUMP OK", CONDUCTIVITY :=, "TANK TEMP" :=, "TEMP IN" :=, "TEMP OUT" :=, "TANK DATA" := "HMI DB".RECUP, "INLET 1 OPEN" => #RECUP."INLET 1 OPEN", "INLET 2 OPEN" => #RECUP."INLET 2 OPEN", "OUTLET OPEN" => #RECUP."OUTLE OPEN", CIRCULATION =>, "START DOZING" => #RECUP."START DOZING", FLUSH => #RECUP.FLUSH, HEATING => #RECUP.HEATING, "PREP DONE" => #RECUP."PREP DONE", "CIP STEP DONE" =>, STATUS =>)
   END_RUNG
   RUNG wire#powerrail
      I_Contact( "IO_MAP".D_OUT."BFV 12" )
   END_RUNG wire#w1
   RUNG wire#powerrail
      Contact( #"ACID CIP START" )
      wire#w2
      { S7_Templates := "SrcType := Real" } LE_Contact(in1 := "HMI DB"."ANALOG VALUES".CONDCTIVITY, in2 := "HMI DB"."COMMON SETPOINTS"."COND MIN FOR RECUP")
      wire#w3
      I_Contact( "IO_MAP".D_IN."RECUPARATION TANK HL" )
      I_Contact( "IO_MAP".D_OUT."BFV 12" )
   END_RUNG wire#w4
   RUNG wire#powerrail
      Contact( #"CAUSTIC CIP START" )
   END_RUNG wire#w2
   RUNG wire#powerrail
      I_Contact( #"WATER FLUSH".Q )
      Contact( #"WATER FLUSH CIP START" )
   END_RUNG wire#w3
   RUNG wire#powerrail
      Contact( #"HOT WTR CIP START" )
      Contact( #"HOT WATER TANK".CIRCULATION )
      { S7_Templates := "SrcType := Real" } LE_Contact(in1 := "HMI DB"."ANALOG VALUES"."RETURN LINE TEMP", in2 := "HMI DB"."COMMON SETPOINTS"."TMP MIN FOR RECUP")
      I_Contact( #"HOT WATER TANK"."INLET 2 OPEN" )
   END_RUNG wire#w3
   // the same network as SCL:
   #"RECUP TANK"(HL := "IO_MAP".D_IN."RECUPARATION TANK HL",   // "TANK"
                 LL := "IO_MAP".D_IN."RECUPARATION TANK LL",
                 "START PREPERATION" := #"RECUP PREP START",
                 "START CIP" := #"RECUP CIP START",
                 "DRAIN COMPLETE" := NOT "IO_MAP".D_OUT."BFV 12",
                 "CHECK TEMP" := FALSE,
                 "CHECK COND" := FALSE,
                 INTERLOCK := false,
                 "INLET 2 CTRL" := (((#"ACID CIP START" OR #"CAUSTIC CIP START") AND ("HMI DB"."ANALOG VALUES".CONDCTIVITY <= "HMI DB"."COMMON SETPOINTS"."COND MIN FOR RECUP")) OR (NOT #"WATER FLUSH".Q AND #"WATER FLUSH CIP START") OR (#"HOT WTR CIP START" AND #"HOT WATER TANK".CIRCULATION AND ("HMI DB"."ANALOG VALUES"."RETURN LINE TEMP" <= "HMI DB"."COMMON SETPOINTS"."TMP MIN FOR RECUP") AND NOT #"HOT WATER TANK"."INLET 2 OPEN")) AND NOT "IO_MAP".D_IN."RECUPARATION TANK HL" AND NOT "IO_MAP".D_OUT."BFV 12",
                 "PUMP OK" := #"PUMP OK",
                 "TANK DATA" := "HMI DB".RECUP,
                 "INLET 1 OPEN" => #RECUP."INLET 1 OPEN",
                 "INLET 2 OPEN" => #RECUP."INLET 2 OPEN",
                 "OUTLET OPEN" => #RECUP."OUTLE OPEN",
                 "START DOZING" => #RECUP."START DOZING",
                 FLUSH => #RECUP.FLUSH,
                 HEATING => #RECUP.HEATING,
                 "PREP DONE" => #RECUP."PREP DONE");
END_REGION

REGION Network 5: RECUP DONE STATUS SAVE
   RUNG wire#powerrail
      Contact( #"RECUP TANK"."PREP DONE" )
      S_Coil( #"RECUP PREP DONE" )
   END_RUNG
   RUNG wire#powerrail
      Contact( #"RECUP TANK"."CIP STEP DONE" )
      wire#w1
      Contact( #"RECUP CIP DONE"[0] )
      Contact( #"RECUP CIP DONE"[1] )
      Contact( #"RECUP CIP DONE"[2] )
      Contact( #"RECUP CIP DONE"[3] )
      S_Coil( #"RECUP CIP DONE"[4] )
   END_RUNG
   RUNG wire#w1
      Contact( #"RECUP CIP DONE"[0] )
      Contact( #"RECUP CIP DONE"[1] )
      Contact( #"RECUP CIP DONE"[2] )
      S_Coil( #"RECUP CIP DONE"[3] )
   END_RUNG
   RUNG wire#w1
      Contact( #"RECUP CIP DONE"[0] )
      Contact( #"RECUP CIP DONE"[1] )
      S_Coil( #"RECUP CIP DONE"[2] )
   END_RUNG
   RUNG wire#w1
      Contact( #"RECUP CIP DONE"[0] )
      S_Coil( #"RECUP CIP DONE"[1] )
   END_RUNG
   RUNG wire#w1
      S_Coil( #"RECUP CIP DONE"[0] )
   END_RUNG
   // the same network as SCL:
   IF #"RECUP TANK"."PREP DONE" THEN #"RECUP PREP DONE" := TRUE; END_IF;
   IF #"RECUP TANK"."CIP STEP DONE" AND #"RECUP CIP DONE"[0] AND #"RECUP CIP DONE"[1] AND #"RECUP CIP DONE"[2] AND #"RECUP CIP DONE"[3] THEN
       #"RECUP CIP DONE"[4] := TRUE;
   END_IF;
   IF #"RECUP TANK"."CIP STEP DONE" AND #"RECUP CIP DONE"[0] AND #"RECUP CIP DONE"[1] AND #"RECUP CIP DONE"[2] THEN
       #"RECUP CIP DONE"[3] := TRUE;
   END_IF;
   IF #"RECUP TANK"."CIP STEP DONE" AND #"RECUP CIP DONE"[0] AND #"RECUP CIP DONE"[1] THEN
       #"RECUP CIP DONE"[2] := TRUE;
   END_IF;
   IF #"RECUP TANK"."CIP STEP DONE" AND #"RECUP CIP DONE"[0] THEN #"RECUP CIP DONE"[1] := TRUE; END_IF;
   IF #"RECUP TANK"."CIP STEP DONE" THEN #"RECUP CIP DONE"[0] := TRUE; END_IF;
END_REGION

REGION Network 6: HOT WATER
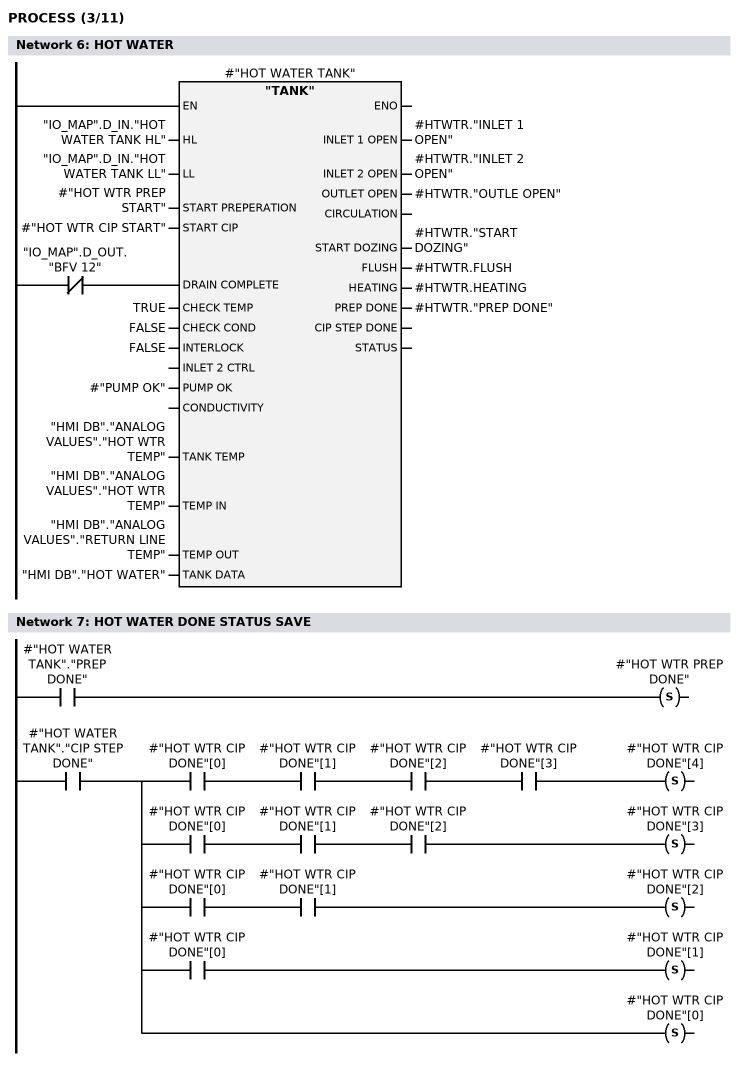
   RUNG wire#powerrail
      #"HOT WATER TANK"("DRAIN COMPLETE" := wire#w1, HL := "IO_MAP".D_IN."HOT WATER TANK HL", LL := "IO_MAP".D_IN."HOT WATER TANK LL", "START PREPERATION" := #"HOT WTR PREP START", "START CIP" := #"HOT WTR CIP START", "CHECK TEMP" := TRUE, "CHECK COND" := FALSE, INTERLOCK := FALSE, "INLET 2 CTRL" :=, "PUMP OK" := #"PUMP OK", CONDUCTIVITY :=, "TANK TEMP" := "HMI DB"."ANALOG VALUES"."HOT WTR TEMP", "TEMP IN" := "HMI DB"."ANALOG VALUES"."HOT WTR TEMP", "TEMP OUT" := "HMI DB"."ANALOG VALUES"."RETURN LINE TEMP", "TANK DATA" := "HMI DB"."HOT WATER", "INLET 1 OPEN" => #HTWTR."INLET 1 OPEN", "INLET 2 OPEN" => #HTWTR."INLET 2 OPEN", "OUTLET OPEN" => #HTWTR."OUTLE OPEN", CIRCULATION =>, "START DOZING" => #HTWTR."START DOZING", FLUSH => #HTWTR.FLUSH, HEATING => #HTWTR.HEATING, "PREP DONE" => #HTWTR."PREP DONE", "CIP STEP DONE" =>, STATUS =>)
   END_RUNG
   RUNG wire#powerrail
      I_Contact( "IO_MAP".D_OUT."BFV 12" )
   END_RUNG wire#w1
   // the same network as SCL:
   #"HOT WATER TANK"(HL := "IO_MAP".D_IN."HOT WATER TANK HL",   // "TANK"
                     LL := "IO_MAP".D_IN."HOT WATER TANK LL",
                     "START PREPERATION" := #"HOT WTR PREP START",
                     "START CIP" := #"HOT WTR CIP START",
                     "DRAIN COMPLETE" := NOT "IO_MAP".D_OUT."BFV 12",
                     "CHECK TEMP" := TRUE,
                     "CHECK COND" := FALSE,
                     INTERLOCK := FALSE,
                     "PUMP OK" := #"PUMP OK",
                     "TANK TEMP" := "HMI DB"."ANALOG VALUES"."HOT WTR TEMP",
                     "TEMP IN" := "HMI DB"."ANALOG VALUES"."HOT WTR TEMP",
                     "TEMP OUT" := "HMI DB"."ANALOG VALUES"."RETURN LINE TEMP",
                     "TANK DATA" := "HMI DB"."HOT WATER",
                     "INLET 1 OPEN" => #HTWTR."INLET 1 OPEN",
                     "INLET 2 OPEN" => #HTWTR."INLET 2 OPEN",
                     "OUTLET OPEN" => #HTWTR."OUTLE OPEN",
                     "START DOZING" => #HTWTR."START DOZING",
                     FLUSH => #HTWTR.FLUSH,
                     HEATING => #HTWTR.HEATING,
                     "PREP DONE" => #HTWTR."PREP DONE");
END_REGION

REGION Network 7: HOT WATER DONE STATUS SAVE
   RUNG wire#powerrail
      Contact( #"HOT WATER TANK"."PREP DONE" )
      S_Coil( #"HOT WTR PREP DONE" )
   END_RUNG
   RUNG wire#powerrail
      Contact( #"HOT WATER TANK"."CIP STEP DONE" )
      wire#w1
      Contact( #"HOT WTR CIP DONE"[0] )
      Contact( #"HOT WTR CIP DONE"[1] )
      Contact( #"HOT WTR CIP DONE"[2] )
      Contact( #"HOT WTR CIP DONE"[3] )
      S_Coil( #"HOT WTR CIP DONE"[4] )
   END_RUNG
   RUNG wire#w1
      Contact( #"HOT WTR CIP DONE"[0] )
      Contact( #"HOT WTR CIP DONE"[1] )
      Contact( #"HOT WTR CIP DONE"[2] )
      S_Coil( #"HOT WTR CIP DONE"[3] )
   END_RUNG
   RUNG wire#w1
      Contact( #"HOT WTR CIP DONE"[0] )
      Contact( #"HOT WTR CIP DONE"[1] )
      S_Coil( #"HOT WTR CIP DONE"[2] )
   END_RUNG
   RUNG wire#w1
      Contact( #"HOT WTR CIP DONE"[0] )
      S_Coil( #"HOT WTR CIP DONE"[1] )
   END_RUNG
   RUNG wire#w1
      S_Coil( #"HOT WTR CIP DONE"[0] )
   END_RUNG
   // the same network as SCL:
   IF #"HOT WATER TANK"."PREP DONE" THEN #"HOT WTR PREP DONE" := TRUE; END_IF;
   IF #"HOT WATER TANK"."CIP STEP DONE" AND #"HOT WTR CIP DONE"[0] AND #"HOT WTR CIP DONE"[1] AND #"HOT WTR CIP DONE"[2] AND #"HOT WTR CIP DONE"[3] THEN
       #"HOT WTR CIP DONE"[4] := TRUE;
   END_IF;
   IF #"HOT WATER TANK"."CIP STEP DONE" AND #"HOT WTR CIP DONE"[0] AND #"HOT WTR CIP DONE"[1] AND #"HOT WTR CIP DONE"[2] THEN
       #"HOT WTR CIP DONE"[3] := TRUE;
   END_IF;
   IF #"HOT WATER TANK"."CIP STEP DONE" AND #"HOT WTR CIP DONE"[0] AND #"HOT WTR CIP DONE"[1] THEN
       #"HOT WTR CIP DONE"[2] := TRUE;
   END_IF;
   IF #"HOT WATER TANK"."CIP STEP DONE" AND #"HOT WTR CIP DONE"[0] THEN
       #"HOT WTR CIP DONE"[1] := TRUE;
   END_IF;
   IF #"HOT WATER TANK"."CIP STEP DONE" THEN #"HOT WTR CIP DONE"[0] := TRUE; END_IF;
END_REGION

REGION Network 8: CAUSTIC TANK
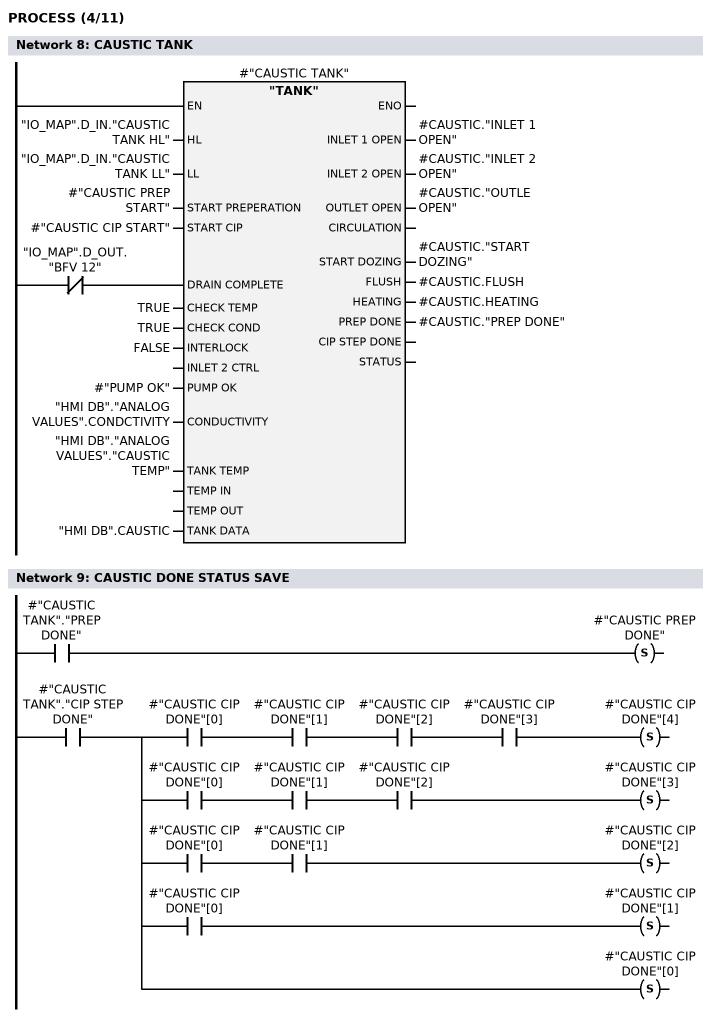
   RUNG wire#powerrail
      #"CAUSTIC TANK"("DRAIN COMPLETE" := wire#w1, HL := "IO_MAP".D_IN."CAUSTIC TANK HL", LL := "IO_MAP".D_IN."CAUSTIC TANK LL", "START PREPERATION" := #"CAUSTIC PREP START", "START CIP" := #"CAUSTIC CIP START", "CHECK TEMP" := TRUE, "CHECK COND" := TRUE, INTERLOCK := FALSE, "INLET 2 CTRL" :=, "PUMP OK" := #"PUMP OK", CONDUCTIVITY := "HMI DB"."ANALOG VALUES".CONDCTIVITY, "TANK TEMP" := "HMI DB"."ANALOG VALUES"."CAUSTIC TEMP", "TEMP IN" :=, "TEMP OUT" :=, "TANK DATA" := "HMI DB".CAUSTIC, "INLET 1 OPEN" => #CAUSTIC."INLET 1 OPEN", "INLET 2 OPEN" => #CAUSTIC."INLET 2 OPEN", "OUTLET OPEN" => #CAUSTIC."OUTLE OPEN", CIRCULATION =>, "START DOZING" => #CAUSTIC."START DOZING", FLUSH => #CAUSTIC.FLUSH, HEATING => #CAUSTIC.HEATING, "PREP DONE" => #CAUSTIC."PREP DONE", "CIP STEP DONE" =>, STATUS =>)
   END_RUNG
   RUNG wire#powerrail
      I_Contact( "IO_MAP".D_OUT."BFV 12" )
   END_RUNG wire#w1
   // the same network as SCL:
   #"CAUSTIC TANK"(HL := "IO_MAP".D_IN."CAUSTIC TANK HL",   // "TANK"
                   LL := "IO_MAP".D_IN."CAUSTIC TANK LL",
                   "START PREPERATION" := #"CAUSTIC PREP START",
                   "START CIP" := #"CAUSTIC CIP START",
                   "DRAIN COMPLETE" := NOT "IO_MAP".D_OUT."BFV 12",
                   "CHECK TEMP" := TRUE,
                   "CHECK COND" := TRUE,
                   INTERLOCK := FALSE,
                   "PUMP OK" := #"PUMP OK",
                   CONDUCTIVITY := "HMI DB"."ANALOG VALUES".CONDCTIVITY,
                   "TANK TEMP" := "HMI DB"."ANALOG VALUES"."CAUSTIC TEMP",
                   "TANK DATA" := "HMI DB".CAUSTIC,
                   "INLET 1 OPEN" => #CAUSTIC."INLET 1 OPEN",
                   "INLET 2 OPEN" => #CAUSTIC."INLET 2 OPEN",
                   "OUTLET OPEN" => #CAUSTIC."OUTLE OPEN",
                   "START DOZING" => #CAUSTIC."START DOZING",
                   FLUSH => #CAUSTIC.FLUSH,
                   HEATING => #CAUSTIC.HEATING,
                   "PREP DONE" => #CAUSTIC."PREP DONE");
END_REGION

REGION Network 9: CAUSTIC DONE STATUS SAVE
   RUNG wire#powerrail
      Contact( #"CAUSTIC TANK"."PREP DONE" )
      S_Coil( #"CAUSTIC PREP DONE" )
   END_RUNG
   RUNG wire#powerrail
      Contact( #"CAUSTIC TANK"."CIP STEP DONE" )
      wire#w1
      Contact( #"CAUSTIC CIP DONE"[0] )
      Contact( #"CAUSTIC CIP DONE"[1] )
      Contact( #"CAUSTIC CIP DONE"[2] )
      Contact( #"CAUSTIC CIP DONE"[3] )
      S_Coil( #"CAUSTIC CIP DONE"[4] )
   END_RUNG
   RUNG wire#w1
      Contact( #"CAUSTIC CIP DONE"[0] )
      Contact( #"CAUSTIC CIP DONE"[1] )
      Contact( #"CAUSTIC CIP DONE"[2] )
      S_Coil( #"CAUSTIC CIP DONE"[3] )
   END_RUNG
   RUNG wire#w1
      Contact( #"CAUSTIC CIP DONE"[0] )
      Contact( #"CAUSTIC CIP DONE"[1] )
      S_Coil( #"CAUSTIC CIP DONE"[2] )
   END_RUNG
   RUNG wire#w1
      Contact( #"CAUSTIC CIP DONE"[0] )
      S_Coil( #"CAUSTIC CIP DONE"[1] )
   END_RUNG
   RUNG wire#w1
      S_Coil( #"CAUSTIC CIP DONE"[0] )
   END_RUNG
   // the same network as SCL:
   IF #"CAUSTIC TANK"."PREP DONE" THEN #"CAUSTIC PREP DONE" := TRUE; END_IF;
   IF #"CAUSTIC TANK"."CIP STEP DONE" AND #"CAUSTIC CIP DONE"[0] AND #"CAUSTIC CIP DONE"[1] AND #"CAUSTIC CIP DONE"[2] AND #"CAUSTIC CIP DONE"[3] THEN
       #"CAUSTIC CIP DONE"[4] := TRUE;
   END_IF;
   IF #"CAUSTIC TANK"."CIP STEP DONE" AND #"CAUSTIC CIP DONE"[0] AND #"CAUSTIC CIP DONE"[1] AND #"CAUSTIC CIP DONE"[2] THEN
       #"CAUSTIC CIP DONE"[3] := TRUE;
   END_IF;
   IF #"CAUSTIC TANK"."CIP STEP DONE" AND #"CAUSTIC CIP DONE"[0] AND #"CAUSTIC CIP DONE"[1] THEN
       #"CAUSTIC CIP DONE"[2] := TRUE;
   END_IF;
   IF #"CAUSTIC TANK"."CIP STEP DONE" AND #"CAUSTIC CIP DONE"[0] THEN #"CAUSTIC CIP DONE"[1] := TRUE; END_IF;
   IF #"CAUSTIC TANK"."CIP STEP DONE" THEN #"CAUSTIC CIP DONE"[0] := TRUE; END_IF;
END_REGION

REGION Network 10: ACIDTANK
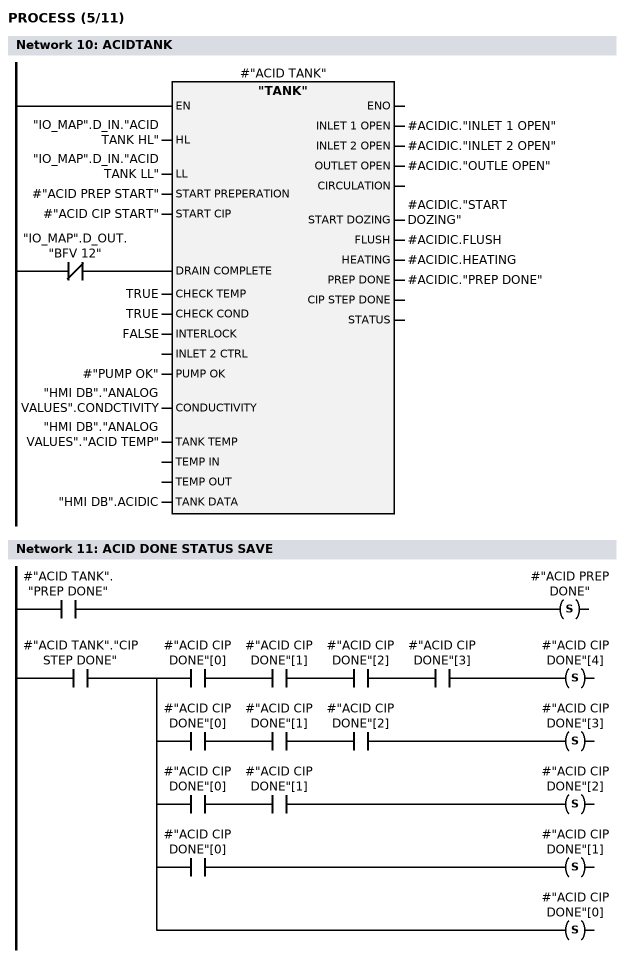
   RUNG wire#powerrail
      #"ACID TANK"("DRAIN COMPLETE" := wire#w1, HL := "IO_MAP".D_IN."ACID TANK HL", LL := "IO_MAP".D_IN."ACID TANK LL", "START PREPERATION" := #"ACID PREP START", "START CIP" := #"ACID CIP START", "CHECK TEMP" := TRUE, "CHECK COND" := TRUE, INTERLOCK := FALSE, "INLET 2 CTRL" :=, "PUMP OK" := #"PUMP OK", CONDUCTIVITY := "HMI DB"."ANALOG VALUES".CONDCTIVITY, "TANK TEMP" := "HMI DB"."ANALOG VALUES"."ACID TEMP", "TEMP IN" :=, "TEMP OUT" :=, "TANK DATA" := "HMI DB".ACIDIC, "INLET 1 OPEN" => #ACIDIC."INLET 1 OPEN", "INLET 2 OPEN" => #ACIDIC."INLET 2 OPEN", "OUTLET OPEN" => #ACIDIC."OUTLE OPEN", CIRCULATION =>, "START DOZING" => #ACIDIC."START DOZING", FLUSH => #ACIDIC.FLUSH, HEATING => #ACIDIC.HEATING, "PREP DONE" => #ACIDIC."PREP DONE", "CIP STEP DONE" =>, STATUS =>)
   END_RUNG
   RUNG wire#powerrail
      I_Contact( "IO_MAP".D_OUT."BFV 12" )
   END_RUNG wire#w1
   // the same network as SCL:
   #"ACID TANK"(HL := "IO_MAP".D_IN."ACID TANK HL",   // "TANK"
                LL := "IO_MAP".D_IN."ACID TANK LL",
                "START PREPERATION" := #"ACID PREP START",
                "START CIP" := #"ACID CIP START",
                "DRAIN COMPLETE" := NOT "IO_MAP".D_OUT."BFV 12",
                "CHECK TEMP" := TRUE,
                "CHECK COND" := TRUE,
                INTERLOCK := FALSE,
                "PUMP OK" := #"PUMP OK",
                CONDUCTIVITY := "HMI DB"."ANALOG VALUES".CONDCTIVITY,
                "TANK TEMP" := "HMI DB"."ANALOG VALUES"."ACID TEMP",
                "TANK DATA" := "HMI DB".ACIDIC,
                "INLET 1 OPEN" => #ACIDIC."INLET 1 OPEN",
                "INLET 2 OPEN" => #ACIDIC."INLET 2 OPEN",
                "OUTLET OPEN" => #ACIDIC."OUTLE OPEN",
                "START DOZING" => #ACIDIC."START DOZING",
                FLUSH => #ACIDIC.FLUSH,
                HEATING => #ACIDIC.HEATING,
                "PREP DONE" => #ACIDIC."PREP DONE");
END_REGION

REGION Network 11: ACID DONE STATUS SAVE
   RUNG wire#powerrail
      Contact( #"ACID TANK"."PREP DONE" )
      S_Coil( #"ACID PREP DONE" )
   END_RUNG
   RUNG wire#powerrail
      Contact( #"ACID TANK"."CIP STEP DONE" )
      wire#w1
      Contact( #"ACID CIP DONE"[0] )
      Contact( #"ACID CIP DONE"[1] )
      Contact( #"ACID CIP DONE"[2] )
      Contact( #"ACID CIP DONE"[3] )
      S_Coil( #"ACID CIP DONE"[4] )
   END_RUNG
   RUNG wire#w1
      Contact( #"ACID CIP DONE"[0] )
      Contact( #"ACID CIP DONE"[1] )
      Contact( #"ACID CIP DONE"[2] )
      S_Coil( #"ACID CIP DONE"[3] )
   END_RUNG
   RUNG wire#w1
      Contact( #"ACID CIP DONE"[0] )
      Contact( #"ACID CIP DONE"[1] )
      S_Coil( #"ACID CIP DONE"[2] )
   END_RUNG
   RUNG wire#w1
      Contact( #"ACID CIP DONE"[0] )
      S_Coil( #"ACID CIP DONE"[1] )
   END_RUNG
   RUNG wire#w1
      S_Coil( #"ACID CIP DONE"[0] )
   END_RUNG
   // the same network as SCL:
   IF #"ACID TANK"."PREP DONE" THEN #"ACID PREP DONE" := TRUE; END_IF;
   IF #"ACID TANK"."CIP STEP DONE" AND #"ACID CIP DONE"[0] AND #"ACID CIP DONE"[1] AND #"ACID CIP DONE"[2] AND #"ACID CIP DONE"[3] THEN
       #"ACID CIP DONE"[4] := TRUE;
   END_IF;
   IF #"ACID TANK"."CIP STEP DONE" AND #"ACID CIP DONE"[0] AND #"ACID CIP DONE"[1] AND #"ACID CIP DONE"[2] THEN
       #"ACID CIP DONE"[3] := TRUE;
   END_IF;
   IF #"ACID TANK"."CIP STEP DONE" AND #"ACID CIP DONE"[0] AND #"ACID CIP DONE"[1] THEN
       #"ACID CIP DONE"[2] := TRUE;
   END_IF;
   IF #"ACID TANK"."CIP STEP DONE" AND #"ACID CIP DONE"[0] THEN #"ACID CIP DONE"[1] := TRUE; END_IF;
   IF #"ACID TANK"."CIP STEP DONE" THEN #"ACID CIP DONE"[0] := TRUE; END_IF;
END_REGION

REGION Network 12: WATER FLUSH STEP
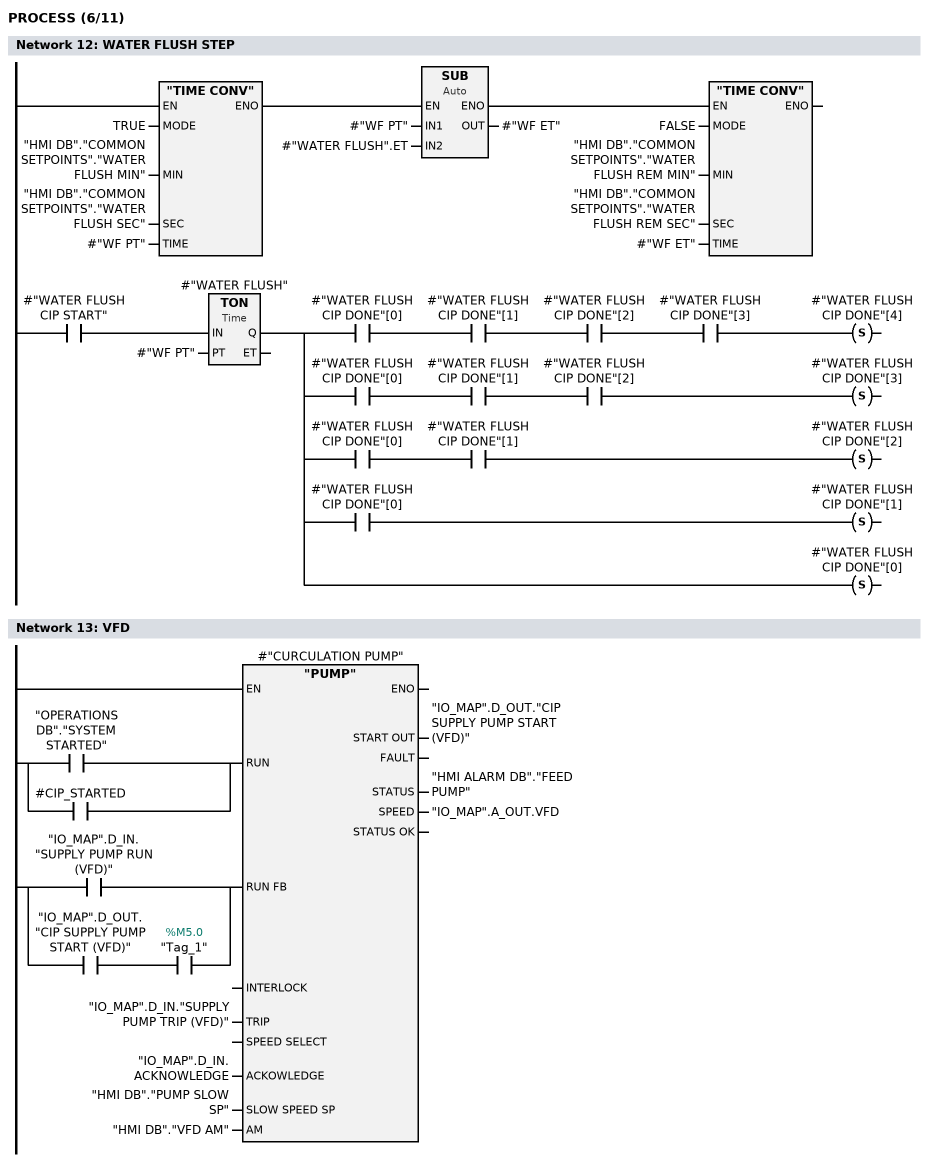
   RUNG wire#powerrail
      "TIME CONV"(MODE := TRUE, MIN := "HMI DB"."COMMON SETPOINTS"."WATER FLUSH MIN", SEC := "HMI DB"."COMMON SETPOINTS"."WATER FLUSH SEC", "TIME" := #"WF PT")
      Sub(in1 := #"WF PT", in2 := #"WATER FLUSH".ET, out => #"WF ET")
      "TIME CONV"(MODE := FALSE, MIN := "HMI DB"."COMMON SETPOINTS"."WATER FLUSH REM MIN", SEC := "HMI DB"."COMMON SETPOINTS"."WATER FLUSH REM SEC", "TIME" := #"WF ET")
   END_RUNG
   RUNG wire#powerrail
      Contact( #"WATER FLUSH CIP START" )
      { S7_Templates := "time_type := Time" } #"WATER FLUSH".TON(pt := #"WF PT", et =>)
      wire#w1
      Contact( #"WATER FLUSH CIP DONE"[0] )
      Contact( #"WATER FLUSH CIP DONE"[1] )
      Contact( #"WATER FLUSH CIP DONE"[2] )
      Contact( #"WATER FLUSH CIP DONE"[3] )
      S_Coil( #"WATER FLUSH CIP DONE"[4] )
   END_RUNG
   RUNG wire#w1
      Contact( #"WATER FLUSH CIP DONE"[0] )
      Contact( #"WATER FLUSH CIP DONE"[1] )
      Contact( #"WATER FLUSH CIP DONE"[2] )
      S_Coil( #"WATER FLUSH CIP DONE"[3] )
   END_RUNG
   RUNG wire#w1
      Contact( #"WATER FLUSH CIP DONE"[0] )
      Contact( #"WATER FLUSH CIP DONE"[1] )
      S_Coil( #"WATER FLUSH CIP DONE"[2] )
   END_RUNG
   RUNG wire#w1
      Contact( #"WATER FLUSH CIP DONE"[0] )
      S_Coil( #"WATER FLUSH CIP DONE"[1] )
   END_RUNG
   RUNG wire#w1
      S_Coil( #"WATER FLUSH CIP DONE"[0] )
   END_RUNG
   // the same network as SCL:
   "TIME CONV"(MODE := TRUE,
               MIN := "HMI DB"."COMMON SETPOINTS"."WATER FLUSH MIN",
               SEC := "HMI DB"."COMMON SETPOINTS"."WATER FLUSH SEC",
               "TIME" := #"WF PT",
               ENO => #_w1);
   IF #_w1 THEN
       #"WF ET" := #"WF PT" - #"WATER FLUSH".ET;
       "TIME CONV"(MODE := FALSE,
                   MIN := "HMI DB"."COMMON SETPOINTS"."WATER FLUSH REM MIN",
                   SEC := "HMI DB"."COMMON SETPOINTS"."WATER FLUSH REM SEC",
                   "TIME" := #"WF ET");
   END_IF;
   #"WATER FLUSH"(IN := #"WATER FLUSH CIP START", PT := #"WF PT");   // TON
   IF #"WATER FLUSH".Q AND #"WATER FLUSH CIP DONE"[0] AND #"WATER FLUSH CIP DONE"[1] AND #"WATER FLUSH CIP DONE"[2] AND #"WATER FLUSH CIP DONE"[3] THEN
       #"WATER FLUSH CIP DONE"[4] := TRUE;
   END_IF;
   IF #"WATER FLUSH".Q AND #"WATER FLUSH CIP DONE"[0] AND #"WATER FLUSH CIP DONE"[1] AND #"WATER FLUSH CIP DONE"[2] THEN
       #"WATER FLUSH CIP DONE"[3] := TRUE;
   END_IF;
   IF #"WATER FLUSH".Q AND #"WATER FLUSH CIP DONE"[0] AND #"WATER FLUSH CIP DONE"[1] THEN
       #"WATER FLUSH CIP DONE"[2] := TRUE;
   END_IF;
   IF #"WATER FLUSH".Q AND #"WATER FLUSH CIP DONE"[0] THEN #"WATER FLUSH CIP DONE"[1] := TRUE; END_IF;
   IF #"WATER FLUSH".Q THEN #"WATER FLUSH CIP DONE"[0] := TRUE; END_IF;
END_REGION

REGION Network 13: VFD
   RUNG wire#powerrail
      #"CURCULATION PUMP"(RUN := wire#w1, "RUN FB" := wire#w2, INTERLOCK :=, TRIP := "IO_MAP".D_IN."SUPPLY PUMP TRIP (VFD)", "SPEED SELECT" :=, ACKOWLEDGE := "IO_MAP".D_IN.ACKNOWLEDGE, "SLOW SPEED SP" := "HMI DB"."PUMP SLOW SP", AM := "HMI DB"."VFD AM", "START OUT" => "IO_MAP".D_OUT."CIP SUPPLY PUMP START (VFD)", FAULT =>, STATUS => "HMI ALARM DB"."FEED PUMP", SPEED => "IO_MAP".A_OUT.VFD, "STATUS OK" =>)
   END_RUNG
   RUNG wire#powerrail
      Contact( "OPERATIONS DB"."SYSTEM STARTED" )
   END_RUNG wire#w1
   RUNG wire#powerrail
      Contact( #CIP_STARTED )
   END_RUNG wire#w1
   RUNG wire#powerrail
      Contact( "IO_MAP".D_IN."SUPPLY PUMP RUN (VFD)" )
   END_RUNG wire#w2
   RUNG wire#powerrail
      Contact( "IO_MAP".D_OUT."CIP SUPPLY PUMP START (VFD)" )
      Contact( "Tag_1" )
   END_RUNG wire#w2
   // the same network as SCL:
   #"CURCULATION PUMP"(RUN := "OPERATIONS DB"."SYSTEM STARTED" OR #CIP_STARTED,   // "PUMP"
                       "RUN FB" := "IO_MAP".D_IN."SUPPLY PUMP RUN (VFD)" OR ("IO_MAP".D_OUT."CIP SUPPLY PUMP START (VFD)" AND "Tag_1"),
                       TRIP := "IO_MAP".D_IN."SUPPLY PUMP TRIP (VFD)",
                       ACKOWLEDGE := "IO_MAP".D_IN.ACKNOWLEDGE,
                       "SLOW SPEED SP" := "HMI DB"."PUMP SLOW SP",
                       AM := "HMI DB"."VFD AM",
                       "START OUT" => "IO_MAP".D_OUT."CIP SUPPLY PUMP START (VFD)",
                       STATUS => "HMI ALARM DB"."FEED PUMP",
                       SPEED => "IO_MAP".A_OUT.VFD);
END_REGION

REGION Network 14: CAUSTIC DOSING
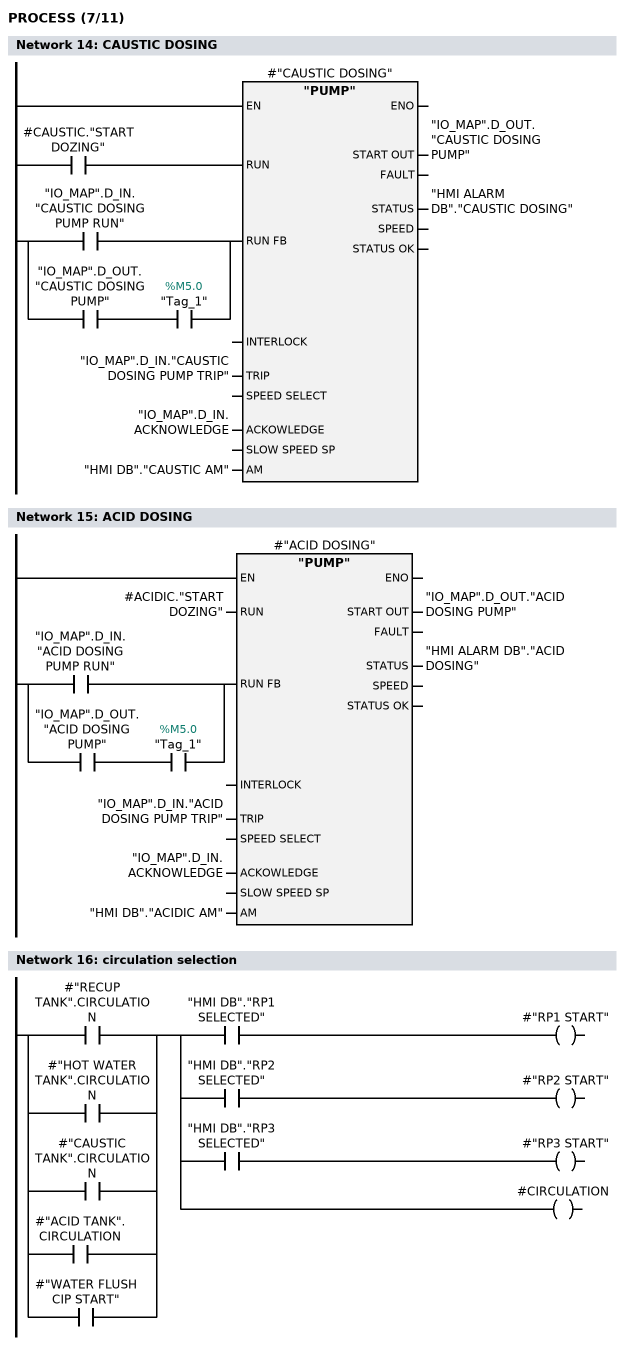
   RUNG wire#powerrail
      #"CAUSTIC DOSING"(RUN := wire#w1, "RUN FB" := wire#w2, INTERLOCK :=, TRIP := "IO_MAP".D_IN."CAUSTIC DOSING PUMP TRIP", "SPEED SELECT" :=, ACKOWLEDGE := "IO_MAP".D_IN.ACKNOWLEDGE, "SLOW SPEED SP" :=, AM := "HMI DB"."CAUSTIC AM", "START OUT" => "IO_MAP".D_OUT."CAUSTIC DOSING PUMP", FAULT =>, STATUS => "HMI ALARM DB"."CAUSTIC DOSING", SPEED =>, "STATUS OK" =>)
   END_RUNG
   RUNG wire#powerrail
      Contact( #CAUSTIC."START DOZING" )
   END_RUNG wire#w1
   RUNG wire#powerrail
      Contact( "IO_MAP".D_IN."CAUSTIC DOSING PUMP RUN" )
   END_RUNG wire#w2
   RUNG wire#powerrail
      Contact( "IO_MAP".D_OUT."CAUSTIC DOSING PUMP" )
      Contact( "Tag_1" )
   END_RUNG wire#w2
   // the same network as SCL:
   #"CAUSTIC DOSING"(RUN := #CAUSTIC."START DOZING",   // "PUMP"
                     "RUN FB" := "IO_MAP".D_IN."CAUSTIC DOSING PUMP RUN" OR ("IO_MAP".D_OUT."CAUSTIC DOSING PUMP" AND "Tag_1"),
                     TRIP := "IO_MAP".D_IN."CAUSTIC DOSING PUMP TRIP",
                     ACKOWLEDGE := "IO_MAP".D_IN.ACKNOWLEDGE,
                     AM := "HMI DB"."CAUSTIC AM",
                     "START OUT" => "IO_MAP".D_OUT."CAUSTIC DOSING PUMP",
                     STATUS => "HMI ALARM DB"."CAUSTIC DOSING");
END_REGION

REGION Network 15: ACID DOSING
   RUNG wire#powerrail
      #"ACID DOSING"("RUN FB" := wire#w1, RUN := #ACIDIC."START DOZING", INTERLOCK :=, TRIP := "IO_MAP".D_IN."ACID DOSING PUMP TRIP", "SPEED SELECT" :=, ACKOWLEDGE := "IO_MAP".D_IN.ACKNOWLEDGE, "SLOW SPEED SP" :=, AM := "HMI DB"."ACIDIC AM", "START OUT" => "IO_MAP".D_OUT."ACID DOSING PUMP", FAULT =>, STATUS => "HMI ALARM DB"."ACID DOSING", SPEED =>, "STATUS OK" =>)
   END_RUNG
   RUNG wire#powerrail
      Contact( "IO_MAP".D_IN."ACID DOSING PUMP RUN" )
   END_RUNG wire#w1
   RUNG wire#powerrail
      Contact( "IO_MAP".D_OUT."ACID DOSING PUMP" )
      Contact( "Tag_1" )
   END_RUNG wire#w1
   // the same network as SCL:
   #"ACID DOSING"(RUN := #ACIDIC."START DOZING",   // "PUMP"
                  "RUN FB" := "IO_MAP".D_IN."ACID DOSING PUMP RUN" OR ("IO_MAP".D_OUT."ACID DOSING PUMP" AND "Tag_1"),
                  TRIP := "IO_MAP".D_IN."ACID DOSING PUMP TRIP",
                  ACKOWLEDGE := "IO_MAP".D_IN.ACKNOWLEDGE,
                  AM := "HMI DB"."ACIDIC AM",
                  "START OUT" => "IO_MAP".D_OUT."ACID DOSING PUMP",
                  STATUS => "HMI ALARM DB"."ACID DOSING");
END_REGION

REGION Network 16: circulation selection
   RUNG wire#powerrail
      Contact( #"RECUP TANK".CIRCULATION )
      wire#w1
      Contact( "HMI DB"."RP1 SELECTED" )
      Coil( #"RP1 START" )
   END_RUNG
   RUNG wire#powerrail
      Contact( #"HOT WATER TANK".CIRCULATION )
   END_RUNG wire#w1
   RUNG wire#powerrail
      Contact( #"CAUSTIC TANK".CIRCULATION )
   END_RUNG wire#w1
   RUNG wire#powerrail
      Contact( #"ACID TANK".CIRCULATION )
   END_RUNG wire#w1
   RUNG wire#powerrail
      Contact( #"WATER FLUSH CIP START" )
   END_RUNG wire#w1
   RUNG wire#w1
      Contact( "HMI DB"."RP2 SELECTED" )
      Coil( #"RP2 START" )
   END_RUNG
   RUNG wire#w1
      Contact( "HMI DB"."RP3 SELECTED" )
      Coil( #"RP3 START" )
   END_RUNG
   RUNG wire#w1
      Coil( #CIRCULATION )
   END_RUNG
   // the same network as SCL:
   #_w1 := #"RECUP TANK".CIRCULATION OR #"HOT WATER TANK".CIRCULATION OR #"CAUSTIC TANK".CIRCULATION OR #"ACID TANK".CIRCULATION OR #"WATER FLUSH CIP START";
   #"RP1 START" := #_w1 AND "HMI DB"."RP1 SELECTED";
   #"RP2 START" := #_w1 AND "HMI DB"."RP2 SELECTED";
   #"RP3 START" := #_w1 AND "HMI DB"."RP3 SELECTED";
   #CIRCULATION := #_w1;
END_REGION

REGION Network 17: RP 1
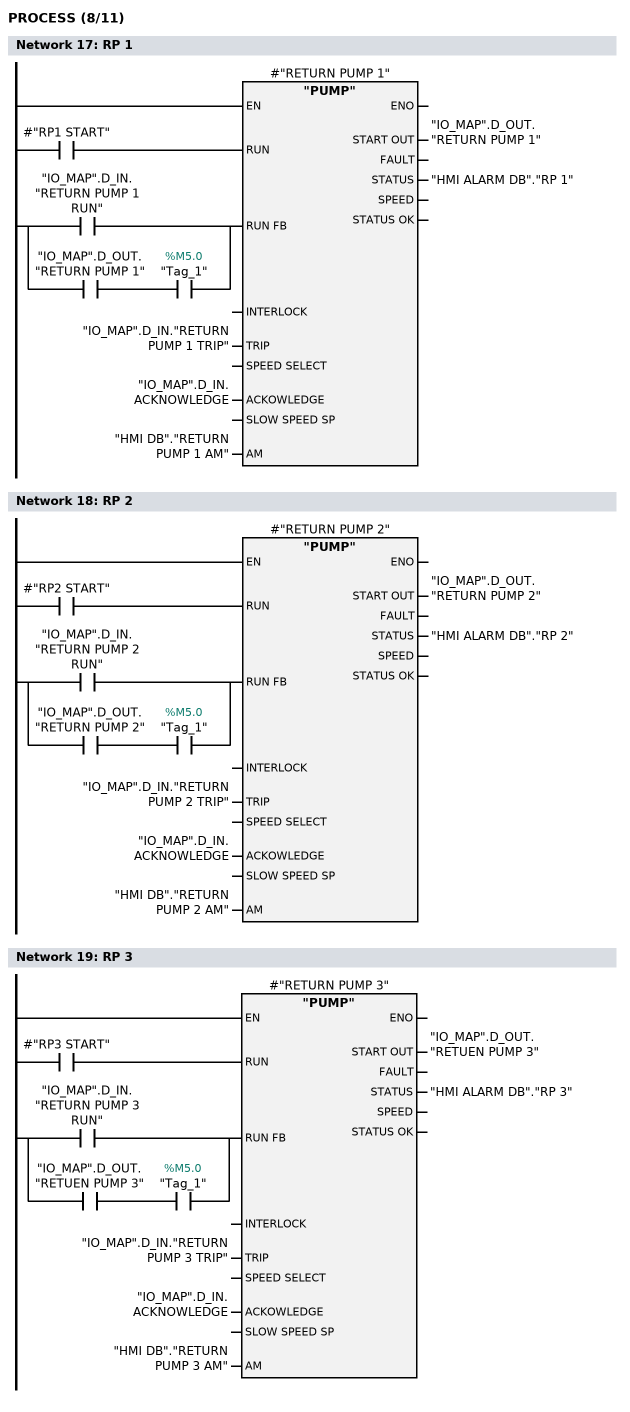
   RUNG wire#powerrail
      #"RETURN PUMP 1"(RUN := wire#w1, "RUN FB" := wire#w2, INTERLOCK :=, TRIP := "IO_MAP".D_IN."RETURN PUMP 1 TRIP", "SPEED SELECT" :=, ACKOWLEDGE := "IO_MAP".D_IN.ACKNOWLEDGE, "SLOW SPEED SP" :=, AM := "HMI DB"."RETURN PUMP 1 AM", "START OUT" => "IO_MAP".D_OUT."RETURN PUMP 1", FAULT =>, STATUS => "HMI ALARM DB"."RP 1", SPEED =>, "STATUS OK" =>)
   END_RUNG
   RUNG wire#powerrail
      Contact( #"RP1 START" )
   END_RUNG wire#w1
   RUNG wire#powerrail
      Contact( "IO_MAP".D_IN."RETURN PUMP 1 RUN" )
   END_RUNG wire#w2
   RUNG wire#powerrail
      Contact( "IO_MAP".D_OUT."RETURN PUMP 1" )
      Contact( "Tag_1" )
   END_RUNG wire#w2
   // the same network as SCL:
   #"RETURN PUMP 1"(RUN := #"RP1 START",   // "PUMP"
                    "RUN FB" := "IO_MAP".D_IN."RETURN PUMP 1 RUN" OR ("IO_MAP".D_OUT."RETURN PUMP 1" AND "Tag_1"),
                    TRIP := "IO_MAP".D_IN."RETURN PUMP 1 TRIP",
                    ACKOWLEDGE := "IO_MAP".D_IN.ACKNOWLEDGE,
                    AM := "HMI DB"."RETURN PUMP 1 AM",
                    "START OUT" => "IO_MAP".D_OUT."RETURN PUMP 1",
                    STATUS => "HMI ALARM DB"."RP 1");
END_REGION

REGION Network 18: RP 2
   RUNG wire#powerrail
      #"RETURN PUMP 2"(RUN := wire#w1, "RUN FB" := wire#w2, INTERLOCK :=, TRIP := "IO_MAP".D_IN."RETURN PUMP 2 TRIP", "SPEED SELECT" :=, ACKOWLEDGE := "IO_MAP".D_IN.ACKNOWLEDGE, "SLOW SPEED SP" :=, AM := "HMI DB"."RETURN PUMP 2 AM", "START OUT" => "IO_MAP".D_OUT."RETURN PUMP 2", FAULT =>, STATUS => "HMI ALARM DB"."RP 2", SPEED =>, "STATUS OK" =>)
   END_RUNG
   RUNG wire#powerrail
      Contact( #"RP2 START" )
   END_RUNG wire#w1
   RUNG wire#powerrail
      Contact( "IO_MAP".D_IN."RETURN PUMP 2 RUN" )
   END_RUNG wire#w2
   RUNG wire#powerrail
      Contact( "IO_MAP".D_OUT."RETURN PUMP 2" )
      Contact( "Tag_1" )
   END_RUNG wire#w2
   // the same network as SCL:
   #"RETURN PUMP 2"(RUN := #"RP2 START",   // "PUMP"
                    "RUN FB" := "IO_MAP".D_IN."RETURN PUMP 2 RUN" OR ("IO_MAP".D_OUT."RETURN PUMP 2" AND "Tag_1"),
                    TRIP := "IO_MAP".D_IN."RETURN PUMP 2 TRIP",
                    ACKOWLEDGE := "IO_MAP".D_IN.ACKNOWLEDGE,
                    AM := "HMI DB"."RETURN PUMP 2 AM",
                    "START OUT" => "IO_MAP".D_OUT."RETURN PUMP 2",
                    STATUS => "HMI ALARM DB"."RP 2");
END_REGION

REGION Network 19: RP 3
   RUNG wire#powerrail
      #"RETURN PUMP 3"(RUN := wire#w1, "RUN FB" := wire#w2, INTERLOCK :=, TRIP := "IO_MAP".D_IN."RETURN PUMP 3 TRIP", "SPEED SELECT" :=, ACKOWLEDGE := "IO_MAP".D_IN.ACKNOWLEDGE, "SLOW SPEED SP" :=, AM := "HMI DB"."RETURN PUMP 3 AM", "START OUT" => "IO_MAP".D_OUT."RETUEN PUMP 3", FAULT =>, STATUS => "HMI ALARM DB"."RP 3", SPEED =>, "STATUS OK" =>)
   END_RUNG
   RUNG wire#powerrail
      Contact( #"RP3 START" )
   END_RUNG wire#w1
   RUNG wire#powerrail
      Contact( "IO_MAP".D_IN."RETURN PUMP 3 RUN" )
   END_RUNG wire#w2
   RUNG wire#powerrail
      Contact( "IO_MAP".D_OUT."RETUEN PUMP 3" )
      Contact( "Tag_1" )
   END_RUNG wire#w2
   // the same network as SCL:
   #"RETURN PUMP 3"(RUN := #"RP3 START",   // "PUMP"
                    "RUN FB" := "IO_MAP".D_IN."RETURN PUMP 3 RUN" OR ("IO_MAP".D_OUT."RETUEN PUMP 3" AND "Tag_1"),
                    TRIP := "IO_MAP".D_IN."RETURN PUMP 3 TRIP",
                    ACKOWLEDGE := "IO_MAP".D_IN.ACKNOWLEDGE,
                    AM := "HMI DB"."RETURN PUMP 3 AM",
                    "START OUT" => "IO_MAP".D_OUT."RETUEN PUMP 3",
                    STATUS => "HMI ALARM DB"."RP 3");
END_REGION

REGION Network 20: BFV CTRL
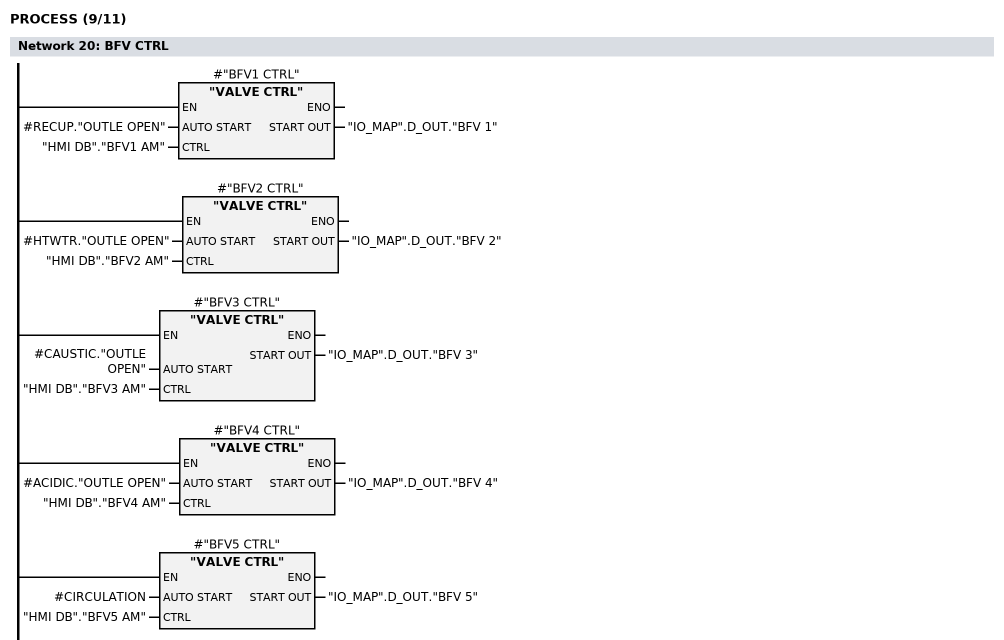
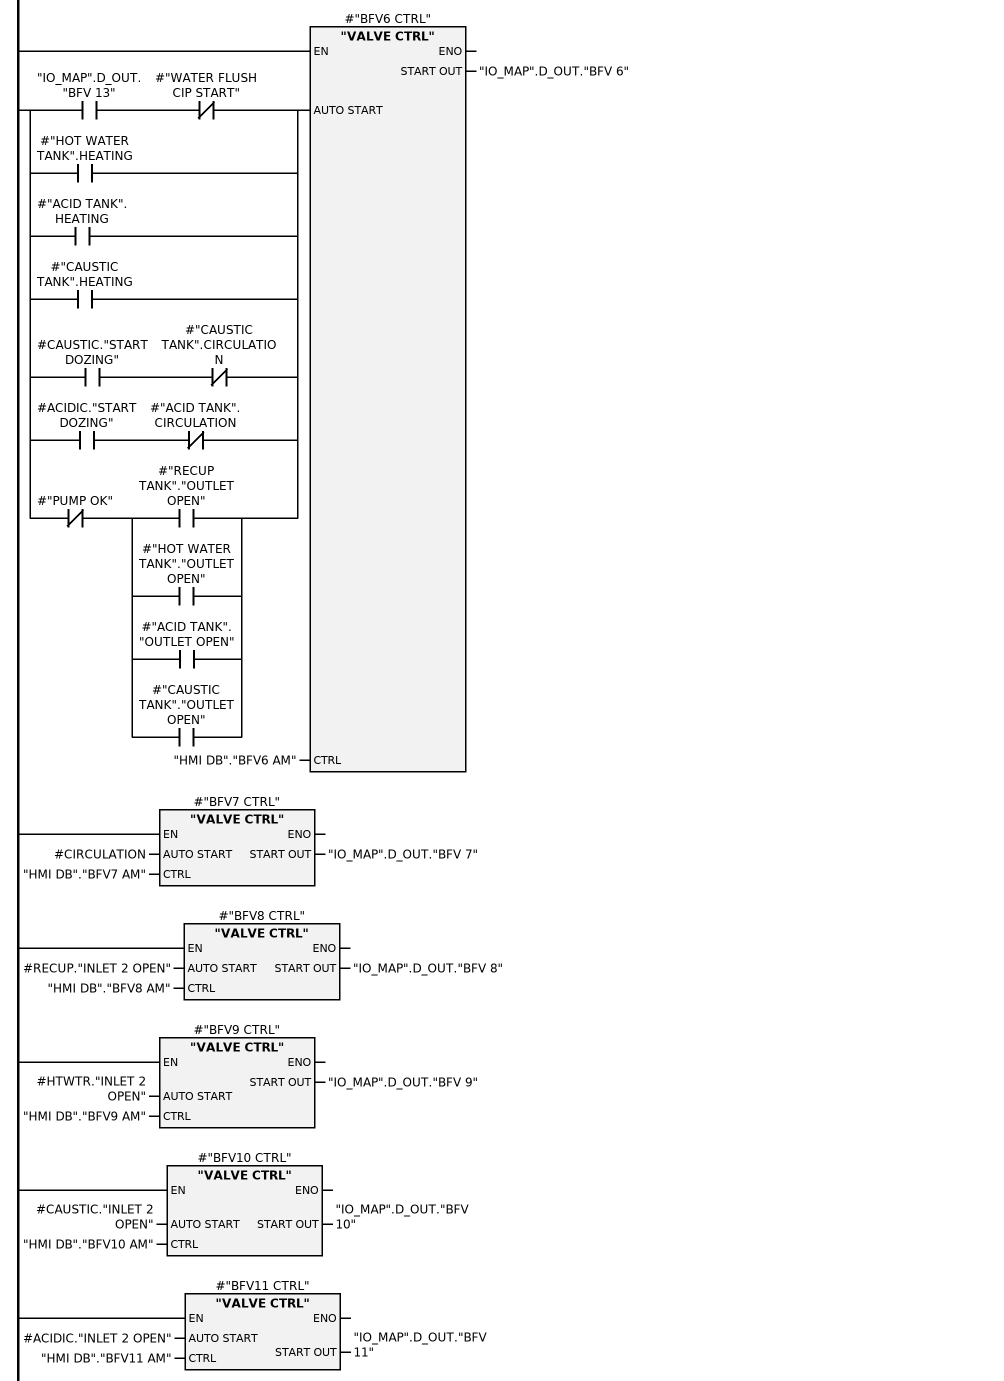
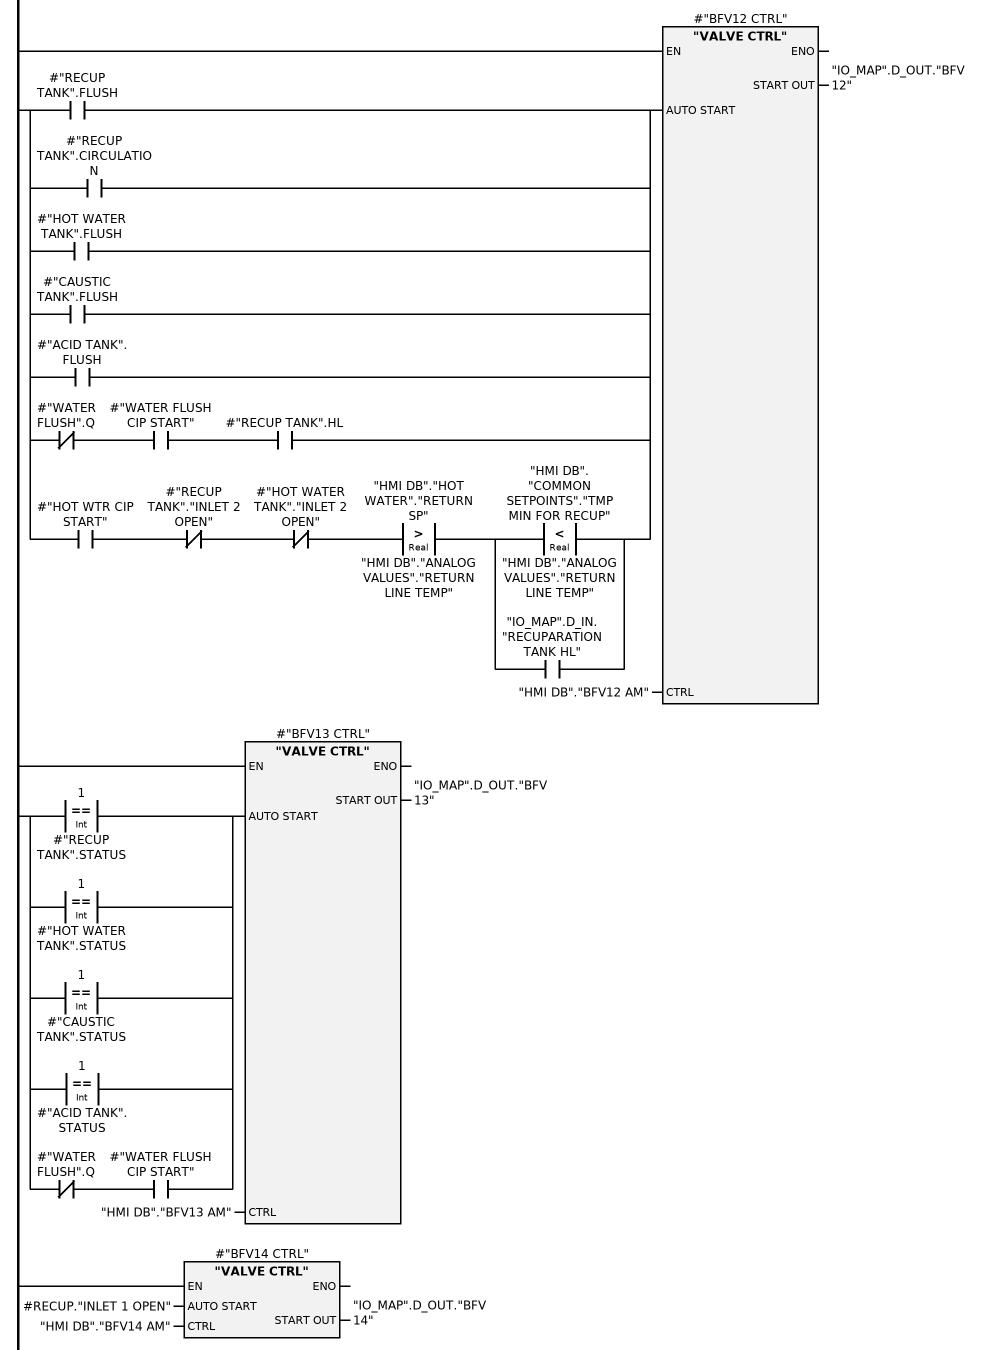
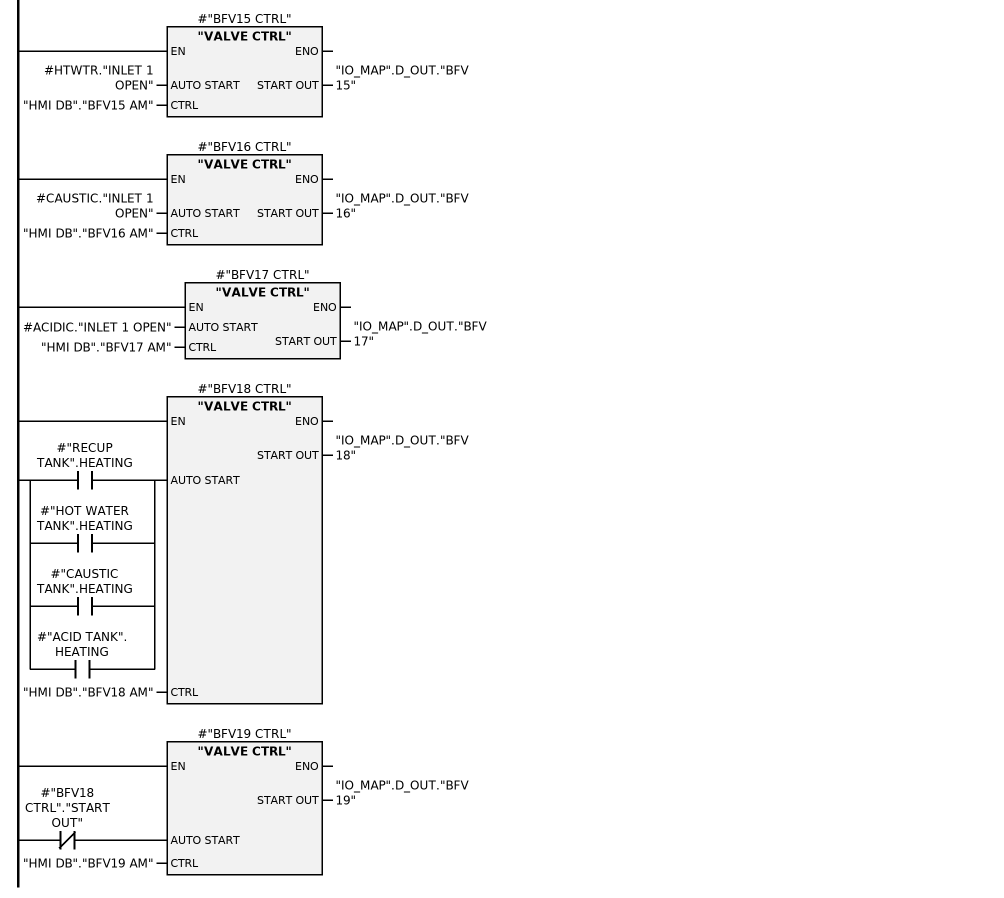
   RUNG wire#powerrail
      #"BFV1 CTRL"("AUTO START" := #RECUP."OUTLE OPEN", CTRL := "HMI DB"."BFV1 AM", "START OUT" => "IO_MAP".D_OUT."BFV 1")
   END_RUNG
   RUNG wire#powerrail
      #"BFV2 CTRL"("AUTO START" := #HTWTR."OUTLE OPEN", CTRL := "HMI DB"."BFV2 AM", "START OUT" => "IO_MAP".D_OUT."BFV 2")
   END_RUNG
   RUNG wire#powerrail
      #"BFV3 CTRL"("AUTO START" := #CAUSTIC."OUTLE OPEN", CTRL := "HMI DB"."BFV3 AM", "START OUT" => "IO_MAP".D_OUT."BFV 3")
   END_RUNG
   RUNG wire#powerrail
      #"BFV4 CTRL"("AUTO START" := #ACIDIC."OUTLE OPEN", CTRL := "HMI DB"."BFV4 AM", "START OUT" => "IO_MAP".D_OUT."BFV 4")
   END_RUNG
   RUNG wire#powerrail
      #"BFV5 CTRL"("AUTO START" := #CIRCULATION, CTRL := "HMI DB"."BFV5 AM", "START OUT" => "IO_MAP".D_OUT."BFV 5")
   END_RUNG
   RUNG wire#powerrail
      #"BFV6 CTRL"("AUTO START" := wire#w2, CTRL := "HMI DB"."BFV6 AM", "START OUT" => "IO_MAP".D_OUT."BFV 6")
   END_RUNG
   RUNG wire#powerrail
      Contact( "IO_MAP".D_OUT."BFV 13" )
      I_Contact( #"WATER FLUSH CIP START" )
   END_RUNG wire#w2
   RUNG wire#powerrail
      Contact( #"HOT WATER TANK".HEATING )
   END_RUNG wire#w2
   RUNG wire#powerrail
      Contact( #"ACID TANK".HEATING )
   END_RUNG wire#w2
   RUNG wire#powerrail
      Contact( #"CAUSTIC TANK".HEATING )
   END_RUNG wire#w2
   RUNG wire#powerrail
      Contact( #CAUSTIC."START DOZING" )
      I_Contact( #"CAUSTIC TANK".CIRCULATION )
   END_RUNG wire#w2
   RUNG wire#powerrail
      Contact( #ACIDIC."START DOZING" )
      I_Contact( #"ACID TANK".CIRCULATION )
   END_RUNG wire#w2
   RUNG wire#powerrail
      I_Contact( #"PUMP OK" )
      wire#w1
      Contact( #"RECUP TANK"."OUTLET OPEN" )
   END_RUNG wire#w2
   RUNG wire#w1
      Contact( #"HOT WATER TANK"."OUTLET OPEN" )
   END_RUNG wire#w2
   RUNG wire#w1
      Contact( #"ACID TANK"."OUTLET OPEN" )
   END_RUNG wire#w2
   RUNG wire#w1
      Contact( #"CAUSTIC TANK"."OUTLET OPEN" )
   END_RUNG wire#w2
   RUNG wire#powerrail
      #"BFV7 CTRL"("AUTO START" := #CIRCULATION, CTRL := "HMI DB"."BFV7 AM", "START OUT" => "IO_MAP".D_OUT."BFV 7")
   END_RUNG
   RUNG wire#powerrail
      #"BFV8 CTRL"("AUTO START" := #RECUP."INLET 2 OPEN", CTRL := "HMI DB"."BFV8 AM", "START OUT" => "IO_MAP".D_OUT."BFV 8")
   END_RUNG
   RUNG wire#powerrail
      #"BFV9 CTRL"("AUTO START" := #HTWTR."INLET 2 OPEN", CTRL := "HMI DB"."BFV9 AM", "START OUT" => "IO_MAP".D_OUT."BFV 9")
   END_RUNG
   RUNG wire#powerrail
      #"BFV10 CTRL"("AUTO START" := #CAUSTIC."INLET 2 OPEN", CTRL := "HMI DB"."BFV10 AM", "START OUT" => "IO_MAP".D_OUT."BFV 10")
   END_RUNG
   RUNG wire#powerrail
      #"BFV11 CTRL"("AUTO START" := #ACIDIC."INLET 2 OPEN", CTRL := "HMI DB"."BFV11 AM", "START OUT" => "IO_MAP".D_OUT."BFV 11")
   END_RUNG
   RUNG wire#powerrail
      #"BFV12 CTRL"("AUTO START" := wire#w4, CTRL := "HMI DB"."BFV12 AM", "START OUT" => "IO_MAP".D_OUT."BFV 12")
   END_RUNG
   RUNG wire#powerrail
      Contact( #"RECUP TANK".FLUSH )
   END_RUNG wire#w4
   RUNG wire#powerrail
      Contact( #"RECUP TANK".CIRCULATION )
   END_RUNG wire#w4
   RUNG wire#powerrail
      Contact( #"HOT WATER TANK".FLUSH )
   END_RUNG wire#w4
   RUNG wire#powerrail
      Contact( #"CAUSTIC TANK".FLUSH )
   END_RUNG wire#w4
   RUNG wire#powerrail
      Contact( #"ACID TANK".FLUSH )
   END_RUNG wire#w4
   RUNG wire#powerrail
      I_Contact( #"WATER FLUSH".Q )
      Contact( #"WATER FLUSH CIP START" )
      Contact( #"RECUP TANK".HL )
   END_RUNG wire#w4
   RUNG wire#powerrail
      Contact( #"HOT WTR CIP START" )
      I_Contact( #"RECUP TANK"."INLET 2 OPEN" )
      I_Contact( #"HOT WATER TANK"."INLET 2 OPEN" )
      { S7_Templates := "SrcType := Real" } GT_Contact(in1 := "HMI DB"."HOT WATER"."RETURN SP", in2 := "HMI DB"."ANALOG VALUES"."RETURN LINE TEMP")
      wire#w3
      { S7_Templates := "SrcType := Real" } LT_Contact(in1 := "HMI DB"."COMMON SETPOINTS"."TMP MIN FOR RECUP", in2 := "HMI DB"."ANALOG VALUES"."RETURN LINE TEMP")
   END_RUNG wire#w4
   RUNG wire#w3
      Contact( "IO_MAP".D_IN."RECUPARATION TANK HL" )
   END_RUNG wire#w4
   RUNG wire#powerrail
      #"BFV13 CTRL"("AUTO START" := wire#w5, CTRL := "HMI DB"."BFV13 AM", "START OUT" => "IO_MAP".D_OUT."BFV 13")
   END_RUNG
   RUNG wire#powerrail
      { S7_Templates := "SrcType := Int" } EQ_Contact(in1 := 1, in2 := #"RECUP TANK".STATUS)
   END_RUNG wire#w5
   RUNG wire#powerrail
      { S7_Templates := "SrcType := Int" } EQ_Contact(in1 := 1, in2 := #"HOT WATER TANK".STATUS)
   END_RUNG wire#w5
   RUNG wire#powerrail
      { S7_Templates := "SrcType := Int" } EQ_Contact(in1 := 1, in2 := #"CAUSTIC TANK".STATUS)
   END_RUNG wire#w5
   RUNG wire#powerrail
      { S7_Templates := "SrcType := Int" } EQ_Contact(in1 := 1, in2 := #"ACID TANK".STATUS)
   END_RUNG wire#w5
   RUNG wire#powerrail
      I_Contact( #"WATER FLUSH".Q )
      Contact( #"WATER FLUSH CIP START" )
   END_RUNG wire#w5
   RUNG wire#powerrail
      #"BFV14 CTRL"("AUTO START" := #RECUP."INLET 1 OPEN", CTRL := "HMI DB"."BFV14 AM", "START OUT" => "IO_MAP".D_OUT."BFV 14")
   END_RUNG
   RUNG wire#powerrail
      #"BFV15 CTRL"("AUTO START" := #HTWTR."INLET 1 OPEN", CTRL := "HMI DB"."BFV15 AM", "START OUT" => "IO_MAP".D_OUT."BFV 15")
   END_RUNG
   RUNG wire#powerrail
      #"BFV16 CTRL"("AUTO START" := #CAUSTIC."INLET 1 OPEN", CTRL := "HMI DB"."BFV16 AM", "START OUT" => "IO_MAP".D_OUT."BFV 16")
   END_RUNG
   RUNG wire#powerrail
      #"BFV17 CTRL"("AUTO START" := #ACIDIC."INLET 1 OPEN", CTRL := "HMI DB"."BFV17 AM", "START OUT" => "IO_MAP".D_OUT."BFV 17")
   END_RUNG
   RUNG wire#powerrail
      #"BFV18 CTRL"("AUTO START" := wire#w6, CTRL := "HMI DB"."BFV18 AM", "START OUT" => "IO_MAP".D_OUT."BFV 18")
   END_RUNG
   RUNG wire#powerrail
      Contact( #"RECUP TANK".HEATING )
   END_RUNG wire#w6
   RUNG wire#powerrail
      Contact( #"HOT WATER TANK".HEATING )
   END_RUNG wire#w6
   RUNG wire#powerrail
      Contact( #"CAUSTIC TANK".HEATING )
   END_RUNG wire#w6
   RUNG wire#powerrail
      Contact( #"ACID TANK".HEATING )
   END_RUNG wire#w6
   RUNG wire#powerrail
      #"BFV19 CTRL"("AUTO START" := wire#w7, CTRL := "HMI DB"."BFV19 AM", "START OUT" => "IO_MAP".D_OUT."BFV 19")
   END_RUNG
   RUNG wire#powerrail
      I_Contact( #"BFV18 CTRL"."START OUT" )
   END_RUNG wire#w7
   // the same network as SCL:
   #"BFV1 CTRL"("AUTO START" := #RECUP."OUTLE OPEN",   // "VALVE CTRL"
                CTRL := "HMI DB"."BFV1 AM",
                "START OUT" => "IO_MAP".D_OUT."BFV 1");
   #"BFV2 CTRL"("AUTO START" := #HTWTR."OUTLE OPEN",   // "VALVE CTRL"
                CTRL := "HMI DB"."BFV2 AM",
                "START OUT" => "IO_MAP".D_OUT."BFV 2");
   #"BFV3 CTRL"("AUTO START" := #CAUSTIC."OUTLE OPEN",   // "VALVE CTRL"
                CTRL := "HMI DB"."BFV3 AM",
                "START OUT" => "IO_MAP".D_OUT."BFV 3");
   #"BFV4 CTRL"("AUTO START" := #ACIDIC."OUTLE OPEN",   // "VALVE CTRL"
                CTRL := "HMI DB"."BFV4 AM",
                "START OUT" => "IO_MAP".D_OUT."BFV 4");
   #"BFV5 CTRL"("AUTO START" := #CIRCULATION, CTRL := "HMI DB"."BFV5 AM", "START OUT" => "IO_MAP".D_OUT."BFV 5");   // "VALVE CTRL"
   #"BFV6 CTRL"("AUTO START" := ("IO_MAP".D_OUT."BFV 13" AND NOT #"WATER FLUSH CIP START") OR #"HOT WATER TANK".HEATING OR #"ACID TANK".HEATING OR #"CAUSTIC TANK".HEATING OR (#CAUSTIC."START DOZING" AND NOT #"CAUSTIC TANK".CIRCULATION) OR (#ACIDIC."START DOZING" AND NOT #"ACID TANK".CIRCULATION) OR (NOT #"PUMP OK" AND (#"RECUP TANK"."OUTLET OPEN" OR #"HOT WATER TANK"."OUTLET OPEN" OR #"ACID TANK"."OUTLET OPEN" OR #"CAUSTIC TANK"."OUTLET OPEN")),   // "VALVE CTRL"
                CTRL := "HMI DB"."BFV6 AM",
                "START OUT" => "IO_MAP".D_OUT."BFV 6");
   #"BFV7 CTRL"("AUTO START" := #CIRCULATION, CTRL := "HMI DB"."BFV7 AM", "START OUT" => "IO_MAP".D_OUT."BFV 7");   // "VALVE CTRL"
   #"BFV8 CTRL"("AUTO START" := #RECUP."INLET 2 OPEN",   // "VALVE CTRL"
                CTRL := "HMI DB"."BFV8 AM",
                "START OUT" => "IO_MAP".D_OUT."BFV 8");
   #"BFV9 CTRL"("AUTO START" := #HTWTR."INLET 2 OPEN",   // "VALVE CTRL"
                CTRL := "HMI DB"."BFV9 AM",
                "START OUT" => "IO_MAP".D_OUT."BFV 9");
   #"BFV10 CTRL"("AUTO START" := #CAUSTIC."INLET 2 OPEN",   // "VALVE CTRL"
                 CTRL := "HMI DB"."BFV10 AM",
                 "START OUT" => "IO_MAP".D_OUT."BFV 10");
   #"BFV11 CTRL"("AUTO START" := #ACIDIC."INLET 2 OPEN",   // "VALVE CTRL"
                 CTRL := "HMI DB"."BFV11 AM",
                 "START OUT" => "IO_MAP".D_OUT."BFV 11");
   #"BFV12 CTRL"("AUTO START" := #"RECUP TANK".FLUSH OR #"RECUP TANK".CIRCULATION OR #"HOT WATER TANK".FLUSH OR #"CAUSTIC TANK".FLUSH OR #"ACID TANK".FLUSH OR (NOT #"WATER FLUSH".Q AND #"WATER FLUSH CIP START" AND #"RECUP TANK".HL) OR (#"HOT WTR CIP START" AND NOT #"RECUP TANK"."INLET 2 OPEN" AND NOT #"HOT WATER TANK"."INLET 2 OPEN" AND ("HMI DB"."HOT WATER"."RETURN SP" > "HMI DB"."ANALOG VALUES"."RETURN LINE TEMP") AND (("HMI DB"."COMMON SETPOINTS"."TMP MIN FOR RECUP" < "HMI DB"."ANALOG VALUES"."RETURN LINE TEMP") OR "IO_MAP".D_IN."RECUPARATION TANK HL")),   // "VALVE CTRL"
                 CTRL := "HMI DB"."BFV12 AM",
                 "START OUT" => "IO_MAP".D_OUT."BFV 12");
   #"BFV13 CTRL"("AUTO START" := (1 = #"RECUP TANK".STATUS) OR (1 = #"HOT WATER TANK".STATUS) OR (1 = #"CAUSTIC TANK".STATUS) OR (1 = #"ACID TANK".STATUS) OR (NOT #"WATER FLUSH".Q AND #"WATER FLUSH CIP START"),   // "VALVE CTRL"
                 CTRL := "HMI DB"."BFV13 AM",
                 "START OUT" => "IO_MAP".D_OUT."BFV 13");
   #"BFV14 CTRL"("AUTO START" := #RECUP."INLET 1 OPEN",   // "VALVE CTRL"
                 CTRL := "HMI DB"."BFV14 AM",
                 "START OUT" => "IO_MAP".D_OUT."BFV 14");
   #"BFV15 CTRL"("AUTO START" := #HTWTR."INLET 1 OPEN",   // "VALVE CTRL"
                 CTRL := "HMI DB"."BFV15 AM",
                 "START OUT" => "IO_MAP".D_OUT."BFV 15");
   #"BFV16 CTRL"("AUTO START" := #CAUSTIC."INLET 1 OPEN",   // "VALVE CTRL"
                 CTRL := "HMI DB"."BFV16 AM",
                 "START OUT" => "IO_MAP".D_OUT."BFV 16");
   #"BFV17 CTRL"("AUTO START" := #ACIDIC."INLET 1 OPEN",   // "VALVE CTRL"
                 CTRL := "HMI DB"."BFV17 AM",
                 "START OUT" => "IO_MAP".D_OUT."BFV 17");
   #"BFV18 CTRL"("AUTO START" := #"RECUP TANK".HEATING OR #"HOT WATER TANK".HEATING OR #"CAUSTIC TANK".HEATING OR #"ACID TANK".HEATING,   // "VALVE CTRL"
                 CTRL := "HMI DB"."BFV18 AM",
                 "START OUT" => "IO_MAP".D_OUT."BFV 18");
   #"BFV19 CTRL"("AUTO START" := NOT #"BFV18 CTRL"."START OUT",   // "VALVE CTRL"
                 CTRL := "HMI DB"."BFV19 AM",
                 "START OUT" => "IO_MAP".D_OUT."BFV 19");
END_REGION

REGION Network 21: SELECTION RESET AFTER CHANGE IN HMI
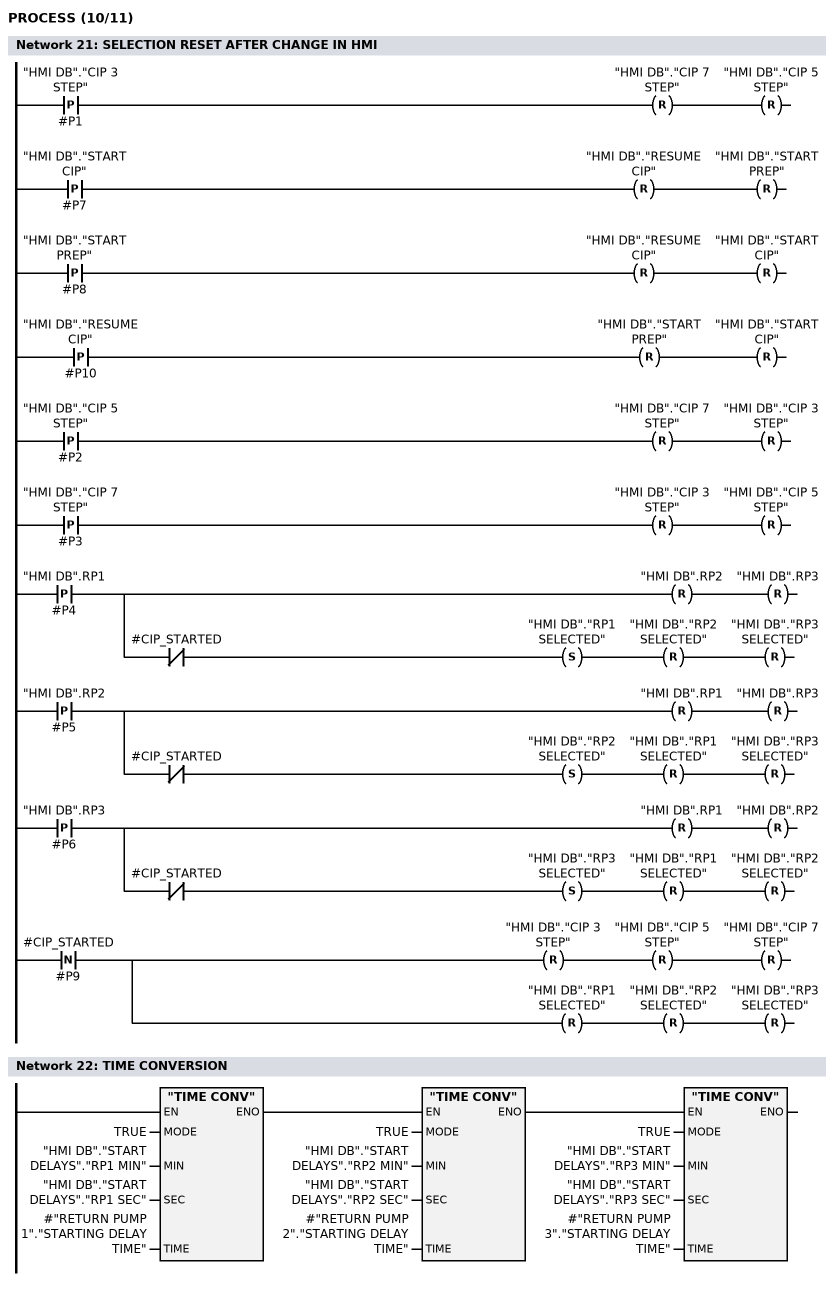
   RUNG wire#powerrail
      P_Contact(operand := "HMI DB"."CIP 3 STEP", bit := #P1)
      R_Coil( "HMI DB"."CIP 7 STEP" )
      R_Coil( "HMI DB"."CIP 5 STEP" )
   END_RUNG
   RUNG wire#powerrail
      P_Contact(operand := "HMI DB"."START CIP", bit := #P7)
      R_Coil( "HMI DB"."RESUME CIP" )
      R_Coil( "HMI DB"."START PREP" )
   END_RUNG
   RUNG wire#powerrail
      P_Contact(operand := "HMI DB"."START PREP", bit := #P8)
      R_Coil( "HMI DB"."RESUME CIP" )
      R_Coil( "HMI DB"."START CIP" )
   END_RUNG
   RUNG wire#powerrail
      P_Contact(operand := "HMI DB"."RESUME CIP", bit := #P10)
      R_Coil( "HMI DB"."START PREP" )
      R_Coil( "HMI DB"."START CIP" )
   END_RUNG
   RUNG wire#powerrail
      P_Contact(operand := "HMI DB"."CIP 5 STEP", bit := #P2)
      R_Coil( "HMI DB"."CIP 7 STEP" )
      R_Coil( "HMI DB"."CIP 3 STEP" )
   END_RUNG
   RUNG wire#powerrail
      P_Contact(operand := "HMI DB"."CIP 7 STEP", bit := #P3)
      R_Coil( "HMI DB"."CIP 3 STEP" )
      R_Coil( "HMI DB"."CIP 5 STEP" )
   END_RUNG
   RUNG wire#powerrail
      P_Contact(operand := "HMI DB".RP1, bit := #P4)
      wire#w1
      R_Coil( "HMI DB".RP2 )
      R_Coil( "HMI DB".RP3 )
   END_RUNG
   RUNG wire#w1
      I_Contact( #CIP_STARTED )
      S_Coil( "HMI DB"."RP1 SELECTED" )
      R_Coil( "HMI DB"."RP2 SELECTED" )
      R_Coil( "HMI DB"."RP3 SELECTED" )
   END_RUNG
   RUNG wire#powerrail
      P_Contact(operand := "HMI DB".RP2, bit := #P5)
      wire#w2
      R_Coil( "HMI DB".RP1 )
      R_Coil( "HMI DB".RP3 )
   END_RUNG
   RUNG wire#w2
      I_Contact( #CIP_STARTED )
      S_Coil( "HMI DB"."RP2 SELECTED" )
      R_Coil( "HMI DB"."RP1 SELECTED" )
      R_Coil( "HMI DB"."RP3 SELECTED" )
   END_RUNG
   RUNG wire#powerrail
      P_Contact(operand := "HMI DB".RP3, bit := #P6)
      wire#w3
      R_Coil( "HMI DB".RP1 )
      R_Coil( "HMI DB".RP2 )
   END_RUNG
   RUNG wire#w3
      I_Contact( #CIP_STARTED )
      S_Coil( "HMI DB"."RP3 SELECTED" )
      R_Coil( "HMI DB"."RP1 SELECTED" )
      R_Coil( "HMI DB"."RP2 SELECTED" )
   END_RUNG
   RUNG wire#powerrail
      N_Contact(operand := #CIP_STARTED, bit := #P9)
      wire#w4
      R_Coil( "HMI DB"."CIP 3 STEP" )
      R_Coil( "HMI DB"."CIP 5 STEP" )
      R_Coil( "HMI DB"."CIP 7 STEP" )
   END_RUNG
   RUNG wire#w4
      R_Coil( "HMI DB"."RP1 SELECTED" )
      R_Coil( "HMI DB"."RP2 SELECTED" )
      R_Coil( "HMI DB"."RP3 SELECTED" )
   END_RUNG
   // the same network as SCL:
   #_w1 := "HMI DB"."CIP 3 STEP" AND NOT #P1;   // rising edge of "HMI DB"."CIP 3 STEP"
   #P1 := "HMI DB"."CIP 3 STEP";
   IF #_w1 THEN
       "HMI DB"."CIP 7 STEP" := FALSE;
       "HMI DB"."CIP 5 STEP" := FALSE;
   END_IF;
   #_w2 := "HMI DB"."START CIP" AND NOT #P7;   // rising edge of "HMI DB"."START CIP"
   #P7 := "HMI DB"."START CIP";
   IF #_w2 THEN
       "HMI DB"."RESUME CIP" := FALSE;
       "HMI DB"."START PREP" := FALSE;
   END_IF;
   #_w3 := "HMI DB"."START PREP" AND NOT #P8;   // rising edge of "HMI DB"."START PREP"
   #P8 := "HMI DB"."START PREP";
   IF #_w3 THEN
       "HMI DB"."RESUME CIP" := FALSE;
       "HMI DB"."START CIP" := FALSE;
   END_IF;
   #_w4 := "HMI DB"."RESUME CIP" AND NOT #P10;   // rising edge of "HMI DB"."RESUME CIP"
   #P10 := "HMI DB"."RESUME CIP";
   IF #_w4 THEN
       "HMI DB"."START PREP" := FALSE;
       "HMI DB"."START CIP" := FALSE;
   END_IF;
   #_w5 := "HMI DB"."CIP 5 STEP" AND NOT #P2;   // rising edge of "HMI DB"."CIP 5 STEP"
   #P2 := "HMI DB"."CIP 5 STEP";
   IF #_w5 THEN
       "HMI DB"."CIP 7 STEP" := FALSE;
       "HMI DB"."CIP 3 STEP" := FALSE;
   END_IF;
   #_w6 := "HMI DB"."CIP 7 STEP" AND NOT #P3;   // rising edge of "HMI DB"."CIP 7 STEP"
   #P3 := "HMI DB"."CIP 7 STEP";
   IF #_w6 THEN
       "HMI DB"."CIP 3 STEP" := FALSE;
       "HMI DB"."CIP 5 STEP" := FALSE;
   END_IF;
   #_w7 := "HMI DB".RP1 AND NOT #P4;   // rising edge of "HMI DB".RP1
   #P4 := "HMI DB".RP1;
   IF #_w7 THEN
       "HMI DB".RP2 := FALSE;
       "HMI DB".RP3 := FALSE;
   END_IF;
   IF #_w7 AND NOT #CIP_STARTED THEN
       "HMI DB"."RP1 SELECTED" := TRUE;
       "HMI DB"."RP2 SELECTED" := FALSE;
       "HMI DB"."RP3 SELECTED" := FALSE;
   END_IF;
   #_w8 := "HMI DB".RP2 AND NOT #P5;   // rising edge of "HMI DB".RP2
   #P5 := "HMI DB".RP2;
   IF #_w8 THEN
       "HMI DB".RP1 := FALSE;
       "HMI DB".RP3 := FALSE;
   END_IF;
   IF #_w8 AND NOT #CIP_STARTED THEN
       "HMI DB"."RP2 SELECTED" := TRUE;
       "HMI DB"."RP1 SELECTED" := FALSE;
       "HMI DB"."RP3 SELECTED" := FALSE;
   END_IF;
   #_w9 := "HMI DB".RP3 AND NOT #P6;   // rising edge of "HMI DB".RP3
   #P6 := "HMI DB".RP3;
   IF #_w9 THEN
       "HMI DB".RP1 := FALSE;
       "HMI DB".RP2 := FALSE;
   END_IF;
   IF #_w9 AND NOT #CIP_STARTED THEN
       "HMI DB"."RP3 SELECTED" := TRUE;
       "HMI DB"."RP1 SELECTED" := FALSE;
       "HMI DB"."RP2 SELECTED" := FALSE;
   END_IF;
   #_w10 := NOT #CIP_STARTED AND #P9;   // falling edge of #CIP_STARTED
   #P9 := #CIP_STARTED;
   IF #_w10 THEN
       "HMI DB"."CIP 3 STEP" := FALSE;
       "HMI DB"."CIP 5 STEP" := FALSE;
       "HMI DB"."CIP 7 STEP" := FALSE;
       "HMI DB"."RP1 SELECTED" := FALSE;
       "HMI DB"."RP2 SELECTED" := FALSE;
       "HMI DB"."RP3 SELECTED" := FALSE;
   END_IF;
END_REGION

REGION Network 22: TIME CONVERSION
   RUNG wire#powerrail
      "TIME CONV"(MODE := TRUE, MIN := "HMI DB"."START DELAYS"."RP1 MIN", SEC := "HMI DB"."START DELAYS"."RP1 SEC", "TIME" := #"RETURN PUMP 1"."STARTING DELAY TIME")
      "TIME CONV"(MODE := TRUE, MIN := "HMI DB"."START DELAYS"."RP2 MIN", SEC := "HMI DB"."START DELAYS"."RP2 SEC", "TIME" := #"RETURN PUMP 2"."STARTING DELAY TIME")
      "TIME CONV"(MODE := TRUE, MIN := "HMI DB"."START DELAYS"."RP3 MIN", SEC := "HMI DB"."START DELAYS"."RP3 SEC", "TIME" := #"RETURN PUMP 3"."STARTING DELAY TIME")
   END_RUNG
   // the same network as SCL:
   "TIME CONV"(MODE := TRUE,
               MIN := "HMI DB"."START DELAYS"."RP1 MIN",
               SEC := "HMI DB"."START DELAYS"."RP1 SEC",
               "TIME" := #"RETURN PUMP 1"."STARTING DELAY TIME",
               ENO => #_w1);
   "TIME CONV"(EN := #_w1,
               MODE := TRUE,
               MIN := "HMI DB"."START DELAYS"."RP2 MIN",
               SEC := "HMI DB"."START DELAYS"."RP2 SEC",
               "TIME" := #"RETURN PUMP 2"."STARTING DELAY TIME",
               ENO => #_w2);
   IF #_w2 THEN
       "TIME CONV"(MODE := TRUE,
                   MIN := "HMI DB"."START DELAYS"."RP3 MIN",
                   SEC := "HMI DB"."START DELAYS"."RP3 SEC",
                   "TIME" := #"RETURN PUMP 3"."STARTING DELAY TIME");
   END_IF;
END_REGION

REGION Network 23: PUMP OK STATUS
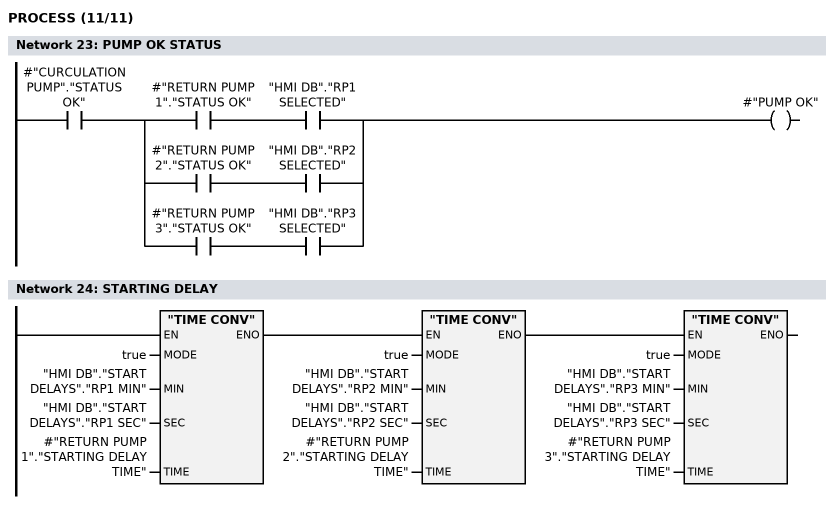
   RUNG wire#powerrail
      Contact( #"CURCULATION PUMP"."STATUS OK" )
      wire#w1
      Contact( #"RETURN PUMP 1"."STATUS OK" )
      Contact( "HMI DB"."RP1 SELECTED" )
      wire#w2
      Coil( #"PUMP OK" )
   END_RUNG
   RUNG wire#w1
      Contact( #"RETURN PUMP 2"."STATUS OK" )
      Contact( "HMI DB"."RP2 SELECTED" )
   END_RUNG wire#w2
   RUNG wire#w1
      Contact( #"RETURN PUMP 3"."STATUS OK" )
      Contact( "HMI DB"."RP3 SELECTED" )
   END_RUNG wire#w2
   // the same network as SCL:
   #"PUMP OK" := #"CURCULATION PUMP"."STATUS OK" AND ((#"RETURN PUMP 1"."STATUS OK" AND "HMI DB"."RP1 SELECTED") OR (#"RETURN PUMP 2"."STATUS OK" AND "HMI DB"."RP2 SELECTED") OR (#"RETURN PUMP 3"."STATUS OK" AND "HMI DB"."RP3 SELECTED"));
END_REGION

REGION Network 24: STARTING DELAY
   RUNG wire#powerrail
      "TIME CONV"(MODE := true, MIN := "HMI DB"."START DELAYS"."RP1 MIN", SEC := "HMI DB"."START DELAYS"."RP1 SEC", "TIME" := #"RETURN PUMP 1"."STARTING DELAY TIME")
      "TIME CONV"(MODE := true, MIN := "HMI DB"."START DELAYS"."RP2 MIN", SEC := "HMI DB"."START DELAYS"."RP2 SEC", "TIME" := #"RETURN PUMP 2"."STARTING DELAY TIME")
      "TIME CONV"(MODE := true, MIN := "HMI DB"."START DELAYS"."RP3 MIN", SEC := "HMI DB"."START DELAYS"."RP3 SEC", "TIME" := #"RETURN PUMP 3"."STARTING DELAY TIME")
   END_RUNG
   // the same network as SCL:
   "TIME CONV"(MODE := true,
               MIN := "HMI DB"."START DELAYS"."RP1 MIN",
               SEC := "HMI DB"."START DELAYS"."RP1 SEC",
               "TIME" := #"RETURN PUMP 1"."STARTING DELAY TIME",
               ENO => #_w1);
   "TIME CONV"(EN := #_w1,
               MODE := true,
               MIN := "HMI DB"."START DELAYS"."RP2 MIN",
               SEC := "HMI DB"."START DELAYS"."RP2 SEC",
               "TIME" := #"RETURN PUMP 2"."STARTING DELAY TIME",
               ENO => #_w2);
   IF #_w2 THEN
       "TIME CONV"(MODE := true,
                   MIN := "HMI DB"."START DELAYS"."RP3 MIN",
                   SEC := "HMI DB"."START DELAYS"."RP3 SEC",
                   "TIME" := #"RETURN PUMP 3"."STARTING DELAY TIME");
   END_IF;
END_REGION

REGION Network 25 (SCL): STATUS DISPLAY ON HMI
   CASE #"CIP_STEP SELECTED" OF

       3:
           "HMI DB"."3 STEP STATUS".%X0:= #"RECUP CIP DONE"[0];
           "HMI DB"."3 STEP STATUS".%X1:= #"HOT WTR CIP DONE"[0];
           "HMI DB"."3 STEP STATUS".%X2:= #"WATER FLUSH CIP DONE"[0];
           "HMI DB"."5 STEP STATUS" := 16#0000;
           "HMI DB"."9 STEP STATUS" := 16#0000;

       5:
           "HMI DB"."5 STEP STATUS".%X0:= #"RECUP CIP DONE"[0];
           "HMI DB"."5 STEP STATUS".%X1:= #"CAUSTIC CIP DONE"[0];
           "HMI DB"."5 STEP STATUS".%X2 := #"WATER FLUSH CIP DONE"[0];
           "HMI DB"."5 STEP STATUS".%X3:= #"HOT WTR CIP DONE"[0];
           "HMI DB"."5 STEP STATUS".%X4:= #"WATER FLUSH CIP DONE"[1];
           "HMI DB"."3 STEP STATUS" := 16#0000;
           "HMI DB"."9 STEP STATUS" := 16#0000;
       9:
           "HMI DB"."9 STEP STATUS".%X0:= #"RECUP CIP DONE"[0];
           "HMI DB"."9 STEP STATUS".%X1:= #"CAUSTIC CIP DONE"[0];
           "HMI DB"."9 STEP STATUS".%X2:= #"WATER FLUSH CIP DONE"[0];
           "HMI DB"."9 STEP STATUS".%X3:= #"ACID CIP DONE"[0];
           "HMI DB"."9 STEP STATUS".%X4:= #"WATER FLUSH CIP DONE"[1];
           "HMI DB"."9 STEP STATUS".%X5:= #"CAUSTIC CIP DONE"[1];
           "HMI DB"."9 STEP STATUS".%X6:= #"WATER FLUSH CIP DONE"[2];
           "HMI DB"."9 STEP STATUS".%X7:= #"HOT WTR CIP DONE"[0];
           "HMI DB"."9 STEP STATUS".%X8:= #"WATER FLUSH CIP DONE"[3];
           "HMI DB"."5 STEP STATUS" := 16#0000;
           "HMI DB"."3 STEP STATUS" := 16#0000;

   END_CASE;
END_REGION
END_FUNCTION_BLOCK

FUNCTION_BLOCK "TANK"
{ S7_Optimized_Access := 'TRUE' }
VERSION : 0.1
   VAR_INPUT 
      HL : Bool;
      LL : Bool;
      "START PREPERATION" : Bool;
      "START CIP" : Bool;
      "DRAIN COMPLETE" : Bool;
      "CHECK TEMP" : Bool;
      "CHECK COND" : Bool;
      INTERLOCK : Bool;
      "INLET 2 CTRL" : Bool;
      "PUMP OK" : Bool;
      CONDUCTIVITY : Real;
      "TANK TEMP" : Real;
      "TEMP IN" : Real;
      "TEMP OUT" : Real;
   END_VAR

   VAR_OUTPUT 
      "INLET 1 OPEN" : Bool;
      "INLET 2 OPEN" : Bool;
      "OUTLET OPEN" : Bool;
      CIRCULATION : Bool;
      "START DOZING" : Bool;
      FLUSH : Bool;
      HEATING : Bool;
      "PREP DONE" : Bool;
      "CIP STEP DONE" : Bool;
      STATUS : Int;
   END_VAR

   VAR_IN_OUT 
      "TANK DATA" : "TANK DATA";
   END_VAR

   VAR 
      "PRIP DONE PULSE" : Bool;
      "START FLUSH" : Bool;
      "FLUSH DELAY" {InstructionName := 'TP_TIME'; LibVersion := '1.0'} : TP_TIME;
      "CIP CYCLE TIME" {InstructionName := 'TONR_TIME'; LibVersion := '1.0'} : TONR_TIME;
   END_VAR

   VAR_TEMP 
      "CIP TIME" : Time;
      "CIP TIME START" : Bool;
      "CIP ET" : Time;
   END_VAR


BEGIN
	
	(*
	STATUS = 0 IDLE
	STATUS = 1 FILLING ONGOING
	STATUS = 2 FILLING FINISHED HEATING STARTED
	STATUS = 3 FILLING FINISHED HEATING AND DOSING STARTED
	STATUS = 5 PREP COMPLETED FILLED
	STATUS = 6 PREP COMPLETED NOT FILLED
	STATUS = 7 PREP COMPLETED HEATED
	STATUS = 8 PREP COMPLETED HEATED AND DOSING COMPLETE
	STATUS = 8 STOPPED DUE TO INTERLOCK FAILURE
	*)
	REGION PREPERATION
	    IF NOT #"START CIP" THEN
	        //RESET OUTPUT WHEN START PREPERATION INPUT IS RESET
	        IF NOT #"START PREPERATION" THEN
	            #STATUS := 0;
	            #"PRIP DONE PULSE" := FALSE;
	            #"PREP DONE" := FALSE;
	            #"INLET 1 OPEN" := FALSE;
	            #"INLET 2 OPEN" := FALSE;
	            #CIRCULATION := FALSE;
	        END_IF;
	        
	        //In the first cycle of START PREPRTATION, if LL is true, it will skip to next step
	        IF #"START PREPERATION" AND NOT #"PRIP DONE PULSE" THEN
	            #"PRIP DONE PULSE" := TRUE;
	            IF #LL THEN
	                IF NOT #"CHECK COND" AND NOT #"CHECK TEMP" THEN
	                    #"PREP DONE" := TRUE;
	                    #STATUS := 6;
	                END_IF;
	            END_IF;
	        END_IF;
	        
	        //if LL is not set, start the valves and motor according to interlock conditions
	        IF #"START PREPERATION" AND (#STATUS = 0 OR #STATUS = 1) AND ((NOT #LL OR #"INLET 1 OPEN") OR #"CHECK TEMP") THEN
	            IF NOT #INTERLOCK THEN
	                #"INLET 1 OPEN" := TRUE;
	                #"START FLUSH" := TRUE;
	                #STATUS := 1;
	                #"INLET 2 OPEN" := #"DRAIN COMPLETE";
	                
	            ELSE
	                #STATUS := 9;
	                #"INLET 1 OPEN" := FALSE;
	                #"INLET 2 OPEN" := FALSE;
	            END_IF;
	        END_IF;
	        
	        //After starting, checking for the HL condition to stop the valves
	        IF #"START PREPERATION" AND #STATUS = 1 THEN
	            IF #HL AND NOT #"CHECK COND" AND NOT #"CHECK TEMP" THEN
	                #STATUS := 5;
	                #"INLET 1 OPEN" := FALSE;
	                #"INLET 2 OPEN" := FALSE;
	                #"PREP DONE" := TRUE;
	            ELSIF #HL AND #"CHECK TEMP" AND NOT #"CHECK COND" THEN
	                #STATUS := 2;
	                #"INLET 1 OPEN" := FALSE;
	                #"INLET 2 OPEN" := FALSE;
	            ELSIF #HL AND #"CHECK TEMP" AND #"CHECK COND" THEN
	                #STATUS := 3;
	                #"INLET 1 OPEN" := FALSE;
	                #"INLET 2 OPEN" := FALSE;
	                
	            END_IF;
	        END_IF;
	        //Tank Filled, Heating confitions.
	        IF #"START PREPERATION" AND #STATUS = 2 AND NOT #"CHECK COND" AND #"CHECK TEMP" AND NOT #HEATING THEN
	            #HEATING := TRUE;
	            #"OUTLET OPEN" := TRUE;
	            RESET_TIMER(#"FLUSH DELAY");
	            #"START FLUSH" := TRUE;
	        ELSIF #"START PREPERATION" AND #STATUS = 2 AND NOT #"CHECK COND" AND #"CHECK TEMP" AND #HEATING THEN
	            IF NOT #FLUSH THEN
	                #"INLET 2 OPEN" := TRUE;
	            END_IF;
	        END_IF;
	        
	        IF #"START PREPERATION" AND #STATUS = 2 AND #"TANK TEMP" > #"TANK DATA"."TANK TEMP SP" THEN
	            #STATUS := 7;
	            #"OUTLET OPEN" := FALSE;
	            #"INLET 2 OPEN" := FALSE;
	            #HEATING := FALSE;
	            #"PREP DONE" := TRUE;
	            
	        END_IF;
	        
	        //Tank Filled, Heating and Dosing confitions.
	        IF #"START PREPERATION" AND #STATUS = 3 THEN
	            IF #"CHECK COND" AND #"CHECK TEMP" AND NOT #HEATING AND NOT #"START DOZING" THEN
	                #HEATING := TRUE;
	                #"OUTLET OPEN" := TRUE;
	                RESET_TIMER(#"FLUSH DELAY");
	                #"START FLUSH" := TRUE;
	            ELSIF #"CHECK COND" AND #"CHECK TEMP" AND #HEATING THEN
	                IF NOT #FLUSH THEN
	                    #"INLET 2 OPEN" := TRUE;
	                    #"START DOZING" := TRUE;
	                END_IF;
	            END_IF;
	            
	            IF #"TANK TEMP" > #"TANK DATA"."TANK TEMP SP" THEN
	                #HEATING := FALSE;
	            END_IF;
	            
	            IF #CONDUCTIVITY > #"TANK DATA"."COND SP" THEN
	                #"START DOZING" := FALSE;
	                
	            END_IF;
	            
	            IF #"TANK TEMP" > #"TANK DATA"."TANK TEMP SP" AND #CONDUCTIVITY > #"TANK DATA"."COND SP" THEN
	                #STATUS := 8;
	                #"OUTLET OPEN" := FALSE;
	                #"INLET 2 OPEN" := FALSE;
	                #"PREP DONE" := TRUE;
	            END_IF;
	        END_IF;
	        
	        
	
	    END_IF;
	
	    
	END_REGION
	
	REGION CIP CYCLE
	    IF NOT #"START PREPERATION" THEN
	        IF #"START CIP" THEN
	            //CONDITION FOR RECUPERATION
	            REGION Recuperation cip
	                //CONDITION FOR RECUPERATION
	                IF NOT #"CHECK COND" AND NOT #"CHECK TEMP" AND NOT #"CIP CYCLE TIME".Q THEN
	                    #"INLET 1 OPEN" := (NOT #LL OR #"INLET 1 OPEN") AND NOT #HL;
	                    IF #"INLET 1 OPEN" THEN
	                        #"OUTLET OPEN" := FALSE;
	                        #"START FLUSH" := TRUE;
	                        #"INLET 2 OPEN" := #"DRAIN COMPLETE";
	                        #CIRCULATION := FALSE;
	                        #STATUS := 1;
	                        
	                    ELSE
	                        #"INLET 2 OPEN" := FALSE;
	                        #"OUTLET OPEN" := TRUE;
	                        #CIRCULATION := #"PUMP OK";
	                        #"CIP TIME START" := TRUE;
	                        #STATUS := 0;
	                    END_IF;
	                ELSIF NOT #"CHECK COND" AND NOT #"CHECK TEMP" AND #"CIP CYCLE TIME".Q THEN
	                    #"INLET 1 OPEN" := FALSE;
	                    #"INLET 2 OPEN" := FALSE;
	                    #"OUTLET OPEN" := FALSE;
	                    #CIRCULATION := FALSE;
	                    #"CIP STEP DONE" := TRUE;
	                    RESET_TIMER(#"CIP CYCLE TIME");
	                END_IF;
	                
	            END_REGION
	
	            //CONDITION FOR HOT WATER
	            REGION HOT WATER
	                
	                IF #"CHECK TEMP" AND NOT #"CHECK COND" AND NOT #"CIP CYCLE TIME".Q THEN
	                    #"INLET 1 OPEN" := (NOT #LL OR #"INLET 1 OPEN") AND NOT #HL;
	                    IF #"INLET 1 OPEN" THEN
	                        #"OUTLET OPEN" := FALSE;
	                        #"START FLUSH" := TRUE;
	                        #"INLET 2 OPEN" := #"DRAIN COMPLETE";
	                        #CIRCULATION := FALSE;
	                        #HEATING := TRUE;
	                        #STATUS := 1;
	                    ELSE
	                        #STATUS := 0;
	                        #"OUTLET OPEN" := TRUE;
	                        
	                        //HEATING AND CIP CYCLE TIME SECTION
	                        IF #"TANK DATA"."TANK TEMP SP" - #"TANK DATA"."HYSTERIRIS TEMP" >= #"TANK TEMP" THEN
	                            #HEATING := TRUE;
	                            #CIRCULATION := FALSE;
	                        ELSIF #"TANK DATA"."TANK TEMP SP" + #"TANK DATA"."HYSTERIRIS TEMP" <= #"TANK TEMP" THEN
	                            #HEATING := FALSE;
	                            #CIRCULATION := #"PUMP OK";
	                        ELSIF #"TANK DATA"."TANK TEMP SP" + #"TANK DATA"."HYSTERIRIS TEMP">#"TANK TEMP"
	                            AND #"TANK DATA"."TANK TEMP SP" - #"TANK DATA"."HYSTERIRIS TEMP" < #"TANK TEMP"  AND  NOT #HEATING THEN
	                            #CIRCULATION := #"PUMP OK";
	                       
	                            
	                        END_IF;
	                        
	                        
	                        //RETURN TEMPERATURE SELECTION
	                        IF #"TANK DATA"."RETURN SP" <= #"TEMP OUT" AND #CIRCULATION THEN
	                            #"INLET 2 OPEN" := TRUE;
	                        ELSIF #"TANK DATA"."RETURN SP" > #"TEMP OUT" AND #CIRCULATION THEN
	                            #"INLET 2 OPEN" := FALSE;
	                        ELSIF #HEATING OR (NOT #"PUMP OK" AND #"OUTLET OPEN")  THEN
	                            #"INLET 2 OPEN" := TRUE;
	                        END_IF;
	                        
	                        // CIP TIMER ONLY WORKS WHEN RETURN TEMP> RETURN TEMP SP
	                        #"CIP TIME START" := #CIRCULATION AND #"INLET 2 OPEN" AND #"PUMP OK";
	                      
	                        
	                    END_IF;
	                ELSIF #"CHECK TEMP" AND NOT #"CHECK COND" AND #"CIP CYCLE TIME".Q THEN
	                    #"INLET 1 OPEN" := FALSE;
	                    #"INLET 2 OPEN" := FALSE;
	                    #"OUTLET OPEN" := FALSE;
	                    #CIRCULATION := FALSE;
	                    RESET_TIMER(#"CIP CYCLE TIME");
	                    #HEATING := FALSE;
	                    #"CIP STEP DONE" := TRUE;
	                END_IF;
	                END_REGION
	                
	            //CONDITION FOR ACID AND CAUSTIC
	                REGION ACID AND CAUSTIC
	                    IF #"CHECK COND" AND #"CHECK TEMP" AND NOT #"CIP CYCLE TIME".Q THEN
	                        #"INLET 1 OPEN" := (NOT #LL OR #"INLET 1 OPEN") AND NOT #HL;
	                        IF #"INLET 1 OPEN" THEN
	                            #"OUTLET OPEN" := FALSE;
	                            #"START FLUSH" := TRUE;
	                            #"INLET 2 OPEN" := #"DRAIN COMPLETE";
	                            #CIRCULATION := FALSE;
	                            #HEATING := #"DRAIN COMPLETE";
	                            #STATUS := 1;
	                            #"START DOZING" := FALSE;
	                        ELSE
	                            #STATUS := 0;
	                            #"OUTLET OPEN" := TRUE;
	                            
	                            //HEATING AND CIP CYCLE TIME SECTION
	                            IF #"TANK DATA"."TANK TEMP SP" - #"TANK DATA"."HYSTERIRIS TEMP" >= #"TANK TEMP"  AND NOT #CIRCULATION THEN
	                                #HEATING := TRUE;
	                                #CIRCULATION := FALSE;
	                                #"INLET 2 OPEN" := TRUE;
	                            ELSIF #"TANK DATA"."TANK TEMP SP" + #"TANK DATA"."HYSTERIRIS TEMP" <= #"TANK TEMP" THEN
	                                #HEATING := FALSE;
	                            END_IF;
	                            //START DOZING BEFORE CIRCULATION
	                            IF #"TANK DATA"."COND SP" - #"TANK DATA"."HYSTERISIS COND" >= #CONDUCTIVITY AND NOT #CIRCULATION THEN
	                                #"START DOZING" := TRUE;
	                                #CIRCULATION := FALSE;
	                                
	                            ELSIF #"TANK DATA"."COND SP" + #"TANK DATA"."HYSTERISIS COND" <= #CONDUCTIVITY THEN
	                                #"START DOZING" := FALSE;
	                            END_IF;
	                            
	                            #CIRCULATION := NOT #HEATING AND  (NOT #"START DOZING" OR #CIRCULATION) AND #"PUMP OK";
	                            
	                            #"CIP TIME START":=#CIRCULATION AND #"TANK DATA"."COND SP" - #"TANK DATA"."HYSTERISIS COND" < #CONDUCTIVITY AND #"PUMP OK" ;
	                            //DOZING WHILE CIRCULATION
	                            IF #CIRCULATION AND #"TANK DATA"."COND SP" - #"TANK DATA"."HYSTERISIS COND" > #CONDUCTIVITY THEN
	                                #"START DOZING" := TRUE;
	                            ELSIF #CIRCULATION AND #"TANK DATA"."COND SP" + #"TANK DATA"."HYSTERISIS COND" < #CONDUCTIVITY THEN
	                                #"START DOZING" := FALSE;
	                            END_IF;
	                                
	                            IF #"TANK DATA"."RETURN SP" <= #CONDUCTIVITY AND #CIRCULATION THEN
	                                #"INLET 2 OPEN" := TRUE;
	                            ELSIF #"TANK DATA"."RETURN SP" > #CONDUCTIVITY AND #CIRCULATION THEN
	                                #"INLET 2 OPEN" := FALSE;
	                            ELSIF #HEATING OR #"START DOZING" THEN
	                                #"INLET 2 OPEN" := TRUE;
	                            END_IF;
	                            
	                           
	                        END_IF;
	                        
	                        
	                    ELSIF #"CHECK TEMP" AND #"CHECK COND" AND #"CIP CYCLE TIME".Q THEN
	                        #"INLET 1 OPEN" := FALSE;
	                        #"INLET 2 OPEN" := FALSE;
	                        #"OUTLET OPEN" := FALSE;
	                        RESET_TIMER(#"CIP CYCLE TIME");
	                        #HEATING := FALSE;
	                        #"CIP STEP DONE" := TRUE;
	                    END_IF;
	                END_REGION
	
	            ELSE
	                #"INLET 1 OPEN" := FALSE;
	                #"INLET 2 OPEN" := FALSE;
	                #"OUTLET OPEN" := FALSE;
	                #CIRCULATION := FALSE;
	                #"START DOZING" := FALSE;
	                #FLUSH := FALSE;
	                #HEATING := FALSE;
	                #"CIP STEP DONE" := FALSE;
	                
	            END_IF;
	     
	        END_IF;
	  
	    
	    
	END_REGION
	
	//CONTROL FOR INLET FROM OUTSIDE WHEN THE CYCLE IS NOT SELECTED ON THIS BLOCK
	REGION INLET 2 CONTROL FORMS OUTSIDE
	    IF NOT #"START CIP" AND NOT #"START PREPERATION" AND #"INLET 2 CTRL" THEN
	        #"INLET 2 OPEN" := TRUE;
	        ELSIF NOT #"START CIP" AND NOT #"START PREPERATION" AND NOT #"INLET 2 CTRL" THEN
	        #"INLET 2 OPEN" := FALSE;
	    END_IF;
	    
	END_REGION
	
	//TIMERS USED. THEY ARE ENABLED FROM BITS CONROLLED FROM THE PROGRAM ABOVE
	REGION TIMERS
	    //timer outside the IF CONDITIONS
	    
	    #"FLUSH DELAY"(IN := #"START FLUSH",
	                   PT := T#15S,
	                   Q => #"FLUSH"); 
	    
	    #"START FLUSH" := #"FLUSH DELAY".Q;
	    "TIME CONV"(MODE := TRUE,
	                MIN := #"TANK DATA"."CYCLE TIME MIN",
	                SEC := #"TANK DATA"."CYCLE TIME SEC",
	                "TIME" := #"CIP TIME");
	    
	    #"CIP CYCLE TIME"(IN := #"CIP TIME START",
	                      PT := #"CIP TIME");
	    #"CIP ET" := #"CIP TIME" - #"CIP CYCLE TIME".ET;
	    "TIME CONV"(MODE := FALSE,
	                MIN := #"TANK DATA"."ELAPSED MIN",
	                SEC := #"TANK DATA"."ELAPSED SEC",
	                "TIME" := #"CIP ET");
	    IF #"CIP CYCLE TIME".Q THEN
	        #"CIP TIME START" := false;
	        // Statement section IF
	        ;
	    END_IF;
	    
	    
	END_REGION
	
	
	
	
	
END_FUNCTION_BLOCK

FUNCTION "TIME CONV" : Void   // FC3, LAD
{ S7_Optimized_Access := 'TRUE' }
VERSION : 0.1
// stored: AutoNumber true, IsIECCheckEnabled false, SetENOAutomatically false, UDAEnableTagReadback false
   VAR_INPUT
      MODE : Bool;
   END_VAR
   VAR_IN_OUT
      MIN : Int;
      SEC : Int;
      "TIME" : Time;
   END_VAR
   VAR_TEMP
      "MUL VAL" : DInt;
   END_VAR
BEGIN

REGION Network 1 (SCL)
   IF #MODE THEN
       #"MUL VAL" := INT_TO_DINT(#SEC + #MIN*60);
       #"MUL VAL" := #"MUL VAL" * 1000;
       #TIME := DINT_TO_TIME( #"MUL VAL");
   ELSIF NOT #MODE THEN
       #MIN := DINT_TO_INT(((TIME_TO_DINT(#TIME) /1000)/60));
       #SEC := DINT_TO_INT(((TIME_TO_DINT(#TIME)/ 1000 MOD 60)));
   END_IF;
END_REGION
END_FUNCTION

FUNCTION_BLOCK "PUMP"
{ S7_Optimized_Access := 'TRUE' }
VERSION : 0.1
   VAR_INPUT 
      RUN : Bool;
      "RUN FB" : Bool;
      INTERLOCK : Bool;
      TRIP : Bool;
      "SPEED SELECT" : Bool;
      ACKOWLEDGE : Bool;
      "SLOW SPEED SP" : Int;
   END_VAR

   VAR_OUTPUT 
      "START OUT" : Bool;
      FAULT : Bool;
      STATUS : Byte;
      SPEED : Int;
      "STATUS OK" : Bool;
   END_VAR

   VAR_IN_OUT 
      AM : "AM CTRL";
   END_VAR

   VAR 
      "RUN FB DELAY" {InstructionName := 'TON_TIME'; LibVersion := '1.0'} : TON_TIME;
      "STARTING DELAY" {InstructionName := 'TON_TIME'; LibVersion := '1.0'} : TON_TIME;
      "STARTING DELAY TIME" { S7_SetPoint := 'True'} : Time;
   END_VAR


BEGIN
	REGION #RUN STOP 
	    //FAULT CONDITION
	    IF (#ACKOWLEDGE) THEN
	        #FAULT := FALSE;
	        #STATUS := 16#0000;
	    END_IF;
	    IF #INTERLOCK OR #TRIP AND (#"START OUT" OR #AM."AUTO/MAN") THEN
	        #FAULT := TRUE;
	        #STATUS.%X0 := #INTERLOCK;
	        #STATUS.%X1 := #TRIP;
	    END_IF;
	    
	    //RUN FEEDBACK CONDITION
	    #"RUN FB DELAY"(IN := #"START OUT" AND NOT #"RUN FB",
	                    PT := T#5S);
	    IF #"RUN FB DELAY".Q THEN
	        #FAULT := TRUE;
	        #STATUS.%X2 := TRUE;
	        
	    END_IF;
	    
	    //RUN CONDITION AUTO
	    #"STARTING DELAY"(IN := #RUN AND #AM."AUTO/MAN" AND NOT #"FAULT",
	                      PT := #"STARTING DELAY TIME");
	    IF #"STARTING DELAY".Q THEN
	        #"START OUT" := TRUE;
	    ELSIF (NOT #RUN AND #AM."AUTO/MAN") OR #FAULT THEN
	        #"START OUT" := FALSE;
	    END_IF;
	    
	    //MOTOR STATUS OK
	    #"STATUS OK" := NOT #TRIP AND #AM."AUTO/MAN" AND NOT #FAULT;
	    
	    // RUN MANUAL
	    IF NOT #AM."AUTO/MAN" THEN
	        #"START OUT" := (#AM."MAN START" OR #"START OUT") AND NOT #AM."MAN STOP" AND NOT #FAULT;
	        
	    END_IF;
	    #AM."MAN START" := FALSE;
	    #AM."MAN STOP" := FALSE;
	END_REGION
	
	REGION #SPEED
	    IF #"START OUT" AND NOT #FAULT THEN
	        IF #"SPEED SELECT" THEN
	            #SPEED := #"SLOW SPEED SP";
	        ELSE
	            #SPEED := 27648;
	        END_IF;
	    ELSE
	        #SPEED := 0;
	    END_IF;
	    
	END_REGION
	
	
END_FUNCTION_BLOCK

FUNCTION_BLOCK "VALVE CTRL"
{ S7_Optimized_Access := 'TRUE' }
VERSION : 0.1
   VAR_INPUT 
      "AUTO START" : Bool;
   END_VAR

   VAR_OUTPUT 
      "START OUT" : Bool;
   END_VAR

   VAR_IN_OUT 
      CTRL : "AM CTRL";
   END_VAR


BEGIN
	//VALVE CONTROL AUTO OR MANUAL BASED ON COMMAND FROM AUTO OR MANUAL
	
	IF #CTRL."AUTO/MAN" THEN
	    #"START OUT" := #"AUTO START";
	ELSIF NOT #CTRL."AUTO/MAN" THEN
	    #"START OUT" := (#"START OUT" OR #CTRL."MAN START") AND NOT #CTRL."MAN STOP";
	    
	END_IF;
	IF #CTRL."MAN START" THEN
	    #CTRL."MAN START" := FALSE;
	END_IF;
	IF #CTRL."MAN STOP" THEN
	    #CTRL."MAN STOP" := FALSE;
	END_IF;
END_FUNCTION_BLOCK

FUNCTION_BLOCK "ALARM"   // FB5, LAD
{ S7_Optimized_Access := 'TRUE' }
VERSION : 0.1
// stored: AutoNumber true, IsIECCheckEnabled false, IsRetainMemResEnabled false, MemoryReserve 100, SetENOAutomatically false, UDAEnableTagReadback false
   VAR
      P1 : Bool;
      P2 : Bool;
      P3 : Bool;
      P4 : Bool;
      P5 : Bool;
      P6 : Bool;
      P7 : Bool;
      P8 : Bool;
      P9 : Bool;
      P10 : Bool;
      P11 : Bool;
      P12 : Bool;
      P13 : Bool;
      P14 : Bool;
      P15 : Bool;
      P16 : Bool;
      P17 : Bool;
      P18 : Bool;
      P19 : Bool;
   END_VAR
   VAR_TEMP   // added for the SCL form of the ladder/FBD networks
      _w1 : Bool;
      _w2 : Bool;
      _w3 : Bool;
      _w4 : Bool;
      _w5 : Bool;
      _w6 : Bool;
      _w7 : Bool;
      _w8 : Bool;
      _w9 : Bool;
      _w10 : Bool;
      _w11 : Bool;
      _w12 : Bool;
      _w13 : Bool;
      _w14 : Bool;
      _w15 : Bool;
      _w16 : Bool;
      _w17 : Bool;
      _w18 : Bool;
   END_VAR
BEGIN

